LIN {X 0,Y 392.045,Z 91.25,A -85,B 0,C 180,E1 -11582.798,E2 -11582.798} C_VEL
LIN {X 0,Y 392.795,Z 97.506,A -85,B 0,C 180,E1 -11584.57,E2 -11584.57} C_VEL
LIN {X 0,Y 391.908,Z 107.771,A -85,B 0,C 180,E1 -11587.322,E2 -11587.322} C_VEL
LIN {X 0,Y 391.284,Z 115.559,A -85,B 0,C 180,E1 -11589.464,E2 -11589.464} C_VEL
LIN {X 0,Y 391.838,Z 118.711,A -85,B 0,C 180,E1 -11589.614,E2 -11589.614} C_VEL
LIN {X 0,Y 396.751,Z 145.759,A -85,B 0,C 180,E1 -11590.385,E2 -11590.385} C_VEL
LIN {X 0,Y 395.854,Z 220.432,A -85,B 0,C 180,E1 -11591.765,E2 -11591.765} C_VEL
LIN {X 0,Y 395.489,Z 230.328,A -85,B 0,C 180,E1 -11592.049,E2 -11592.049} C_VEL
LIN {X 0,Y 394.92,Z 240.302,A -85,B 0,C 180,E1 -11592.457,E2 -11592.457} C_VEL
LIN {X 0,Y 394.307,Z 250.666,A -85,B 0,C 180,E1 -11593.031,E2 -11593.031} C_VEL
LIN {X 0,Y 393.558,Z 259.797,A -85,B 0,C 180,E1 -11593.665,E2 -11593.665} C_VEL
LIN {X 0,Y 392.875,Z 268.795,A -85,B 0,C 180,E1 -11594.435,E2 -11594.435} C_VEL
LIN {X 0,Y 392.089,Z 277.523,A -85,B 0,C 180,E1 -11595.334,E2 -11595.334} C_VEL
LIN {X 0,Y 391.44,Z 285.346,A -85,B 0,C 180,E1 -11596.297,E2 -11596.297} C_VEL
LIN {X 0,Y 390.892,Z 292.141,A -85,B 0,C 180,E1 -11597.276,E2 -11597.276} C_VEL
LIN {X 0,Y 390.295,Z 298.342,A -85,B 0,C 180,E1 -11598.312,E2 -11598.312} C_VEL
LIN {X 0,Y 389.714,Z 304.879,A -85,B 0,C 180,E1 -11599.611,E2 -11599.611} C_VEL
LIN {X 0,Y 389.377,Z 309.381,A -85,B 0,C 180,E1 -11600.651,E2 -11600.651} C_VEL
LIN {X 0,Y 389.017,Z 314.872,A -85,B 0,C 180,E1 -11602.213,E2 -11602.213} C_VEL
LIN {X 0,Y 388.796,Z 319.196,A -85,B 0,C 180,E1 -11603.774,E2 -11603.774} C_VEL
LIN {X 0,Y 388.738,Z 321.563,A -85,B 0,C 180,E1 -11604.814,E2 -11604.814} C_VEL
LIN {X 0,Y 388.7,Z 323.362,A -85,B 0,C 180,E1 -11605.853,E2 -11605.853} C_VEL
LIN {X 0,Y 388.661,Z 325.805,A -85,B 0,C 180,E1 -11607.927,E2 -11607.927} C_VEL
LIN {X 0,Y 388.705,Z 326.395,A -85,B 0,C 180,E1 -11608.964,E2 -11608.964} C_VEL
LIN {X 0,Y 388.705,Z 326.395,A -85,B 0,C 180,E1 -11611.036,E2 -11611.036} C_VEL
LIN {X 0,Y 388.661,Z 325.805,A -85,B 0,C 180,E1 -11612.073,E2 -11612.073} C_VEL
LIN {X 0,Y 388.699,Z 323.362,A -85,B 0,C 180,E1 -11614.147,E2 -11614.147} C_VEL
LIN {X 0,Y 388.726,Z 320.312,A -85,B 0,C 180,E1 -11615.75,E2 -11615.75} C_VEL
LIN {X 0,Y 388.933,Z 316.426,A -85,B 0,C 180,E1 -11617.267,E2 -11617.267} C_VEL
LIN {X 0,Y 389.249,Z 311.297,A -85,B 0,C 180,E1 -11618.828,E2 -11618.828} C_VEL
LIN {X 0,Y 389.628,Z 306.034,A -85,B 0,C 180,E1 -11620.129,E2 -11620.129} C_VEL
LIN {X 0,Y 390.149,Z 299.717,A -85,B 0,C 180,E1 -11621.429,E2 -11621.429} C_VEL
LIN {X 0,Y 390.723,Z 293.767,A -85,B 0,C 180,E1 -11622.465,E2 -11622.465} C_VEL
LIN {X 0,Y 391.336,Z 286.839,A -85,B 0,C 180,E1 -11623.501,E2 -11623.501} C_VEL
LIN {X 0,Y 392.026,Z 278.658,A -85,B 0,C 180,E1 -11624.536,E2 -11624.536} C_VEL
LIN {X 0,Y 392.733,Z 270.146,A -85,B 0,C 180,E1 -11625.438,E2 -11625.438} C_VEL
LIN {X 0,Y 393.459,Z 261.43,A -85,B 0,C 180,E1 -11626.206,E2 -11626.206} C_VEL
LIN {X 0,Y 394.208,Z 251.672,A -85,B 0,C 180,E1 -11626.907,E2 -11626.907} C_VEL
LIN {X 0,Y 394.854,Z 241.59,A -85,B 0,C 180,E1 -11627.479,E2 -11627.479} C_VEL
LIN {X 0,Y 395.411,Z 232.076,A -85,B 0,C 180,E1 -11627.888,E2 -11627.888} C_VEL
LIN {X 0,Y 395.772,Z 221.762,A -85,B 0,C 180,E1 -11628.205,E2 -11628.205} C_VEL
LIN {X 0,Y 396.467,Z 173.837,A -85,B 0,C 180,E1 -11629.102,E2 -11629.102} C_VEL
LIN {X 0,Y 396.69,Z 145.088,A -85,B 0,C 180,E1 -11629.631,E2 -11629.631} C_VEL
LIN {X 0,Y 391.471,Z 116.921,A -85,B 0,C 180,E1 -11630.44,E2 -11630.44} C_VEL
LIN {X 0,Y 391.302,Z 115.351,A -85,B 0,C 180,E1 -11630.57,E2 -11630.57} C_VEL
LIN {X 0,Y 392.552,Z 100.812,A -85,B 0,C 180,E1 -11634.598,E2 -11634.598} C_VEL
LIN {X 0,Y 392.796,Z 95.971,A -85,B 0,C 180,E1 -11635.937,E2 -11635.937} C_VEL
LIN {X 0,Y 391.365,Z 87.664,A -85,B 0,C 180,E1 -11638.366,E2 -11638.366} C_VEL
LIN {X 0,Y 390.091,Z 81.417,A -85,B 0,C 180,E1 -11640.333,E2 -11640.333} C_VEL
LIN {X 0,Y 390.071,Z 81.395,A -85,B 0,C 180,E1 -11644.024,E2 -11644.024} C_VEL
LIN {X 0,Y 390.047,Z 81.402,A -85,B 0,C 180,E1 -11647.551,E2 -11647.551} C_VEL
LIN {X 0,Y 390.058,Z 81.38,A -85,B 0,C 180,E1 -11650.821,E2 -11650.821} C_VEL
LIN {X 0,Y 390.056,Z 81.396,A -85,B 0,C 180,E1 -11653.886,E2 -11653.886} C_VEL
LIN {X 0,Y 390.058,Z 81.396,A -85,B 0,C 180,E1 -11656.789,E2 -11656.789} C_VEL
LIN {X 0,Y 390.058,Z 81.388,A -85,B 0,C 180,E1 -11659.56,E2 -11659.56} C_VEL
LIN {X 0,Y 390.044,Z 81.398,A -85,B 0,C 180,E1 -11662.449,E2 -11662.449} C_VEL
LIN {X 0,Y 390.069,Z 81.38,A -85,B 0,C 180,E1 -11665.975,E2 -11665.975} C_VEL
LIN {X 0,Y 390.048,Z 81.396,A -85,B 0,C 180,E1 -11669.868,E2 -11669.868} C_VEL
LIN {X 0,Y 390.114,Z 81.372,A -85,B 0,C 180,E1 -11673.231,E2 -11673.231} C_VEL
LIN {X 0,Y 390.107,Z 81.393,A -85,B 0,C 180,E1 -11676.75,E2 -11676.75} C_VEL
LIN {X 0,Y 390.105,Z 81.378,A -85,B 0,C 180,E1 -11679.983,E2 -11679.983} C_VEL
LIN {X 0,Y 390.139,Z 81.378,A -85,B 0,C 180,E1 -11683.248,E2 -11683.248} C_VEL
LIN {X 0,Y 390.195,Z 81.377,A -85,B 0,C 180,E1 -11686.561,E2 -11686.561} C_VEL
LIN {X 0,Y 390.205,Z 81.355,A -85,B 0,C 180,E1 -11690.671,E2 -11690.671} C_VEL
LIN {X 0,Y 390.319,Z 81.359,A -85,B 0,C 180,E1 -11692.759,E2 -11692.759} C_VEL
LIN {X 0,Y 390.23,Z 81.374,A -85,B 0,C 180,E1 -11694.833,E2 -11694.833} C_VEL
LIN {X 0,Y 390.418,Z 81.341,A -85,B 0,C 180,E1 -11697.936,E2 -11697.936} C_VEL
LIN {X 0,Y 390.548,Z 81.311,A -85,B 0,C 180,E1 -11699.999,E2 -11699.999} C_VEL
LIN {X 0,Y 390.31,Z 81.358,A -85,B 0,C 180,E1 -11703.096,E2 -11703.096} C_VEL
LIN {X 0,Y 390.309,Z 81.36,A -85,B 0,C 180,E1 -11706.633,E2 -11706.633} C_VEL
LIN {X 0,Y 390.206,Z 81.356,A -85,B 0,C 180,E1 -11709.328,E2 -11709.328} C_VEL
LIN {X 0,Y 390.177,Z 81.375,A -85,B 0,C 180,E1 -11712.482,E2 -11712.482} C_VEL
LIN {X 0,Y 390.139,Z 81.385,A -85,B 0,C 180,E1 -11715.676,E2 -11715.676} C_VEL
LIN {X 0,Y 390.104,Z 81.37,A -85,B 0,C 180,E1 -11718.921,E2 -11718.921} C_VEL
LIN {X 0,Y 390.045,Z 81.395,A -85,B 0,C 180,E1 -11722.233,E2 -11722.233} C_VEL
LIN {X 0,Y 390.117,Z 81.379,A -85,B 0,C 180,E1 -11725.743,E2 -11725.743} C_VEL
LIN {X 0,Y 390.056,Z 81.391,A -85,B 0,C 180,E1 -11729.109,E2 -11729.109} C_VEL
LIN {X 0,Y 390.04,Z 81.396,A -85,B 0,C 180,E1 -11732.721,E2 -11732.721} C_VEL
LIN {X 0,Y 390.055,Z 81.391,A -85,B 0,C 180,E1 -11735.825,E2 -11735.825} C_VEL
LIN {X 0,Y 390.071,Z 81.39,A -85,B 0,C 180,E1 -11739.219,E2 -11739.219} C_VEL
LIN {X 0,Y 390.077,Z 81.392,A -85,B 0,C 180,E1 -11742.38,E2 -11742.38} C_VEL
LIN {X 0,Y 390.051,Z 81.378,A -85,B 0,C 180,E1 -11746.114,E2 -11746.114} C_VEL
LIN {X 0,Y 390.052,Z 81.381,A -85,B 0,C 180,E1 -11749.56,E2 -11749.56} C_VEL
LIN {X 0,Y 390.042,Z 81.4,A -85,B 0,C 180,E1 -11752.448,E2 -11752.448} C_VEL
LIN {X 0,Y 390.064,Z 81.374,A -85,B 0,C 180,E1 -11755.975,E2 -11755.975} C_VEL
LIN {X 0,Y 390.035,Z 81.39,A -85,B 0,C 180,E1 -11759.7,E2 -11759.7} C_VEL
LIN {X 0,Y 390.11,Z 81.392,A -85,B 0,C 180,E1 -11763.232,E2 -11763.232} C_VEL
LIN {X 0,Y 390.103,Z 81.393,A -85,B 0,C 180,E1 -11766.75,E2 -11766.75} C_VEL
LIN {X 0,Y 390.1,Z 81.395,A -85,B 0,C 180,E1 -11769.983,E2 -11769.983} C_VEL
LIN {X 0,Y 390.135,Z 81.391,A -85,B 0,C 180,E1 -11773.248,E2 -11773.248} C_VEL
LIN {X 0,Y 390.191,Z 81.383,A -85,B 0,C 180,E1 -11776.561,E2 -11776.561} C_VEL
LIN {X 0,Y 390.202,Z 81.382,A -85,B 0,C 180,E1 -11780.671,E2 -11780.671} C_VEL
LIN {X 0,Y 390.404,Z 81.767,A -85,B 0,C 180,E1 -11781.927,E2 -11781.927} C_VEL
LIN {X 0,Y 391.193,Z 83.981,A -85,B 0,C 180,E1 -11782.905,E2 -11782.905} C_VEL
LIN {X 0,Y 392.561,Z 85.719,A -85,B 0,C 180,E1 -11783.962,E2 -11783.962} C_VEL
LIN {X 0,Y 394.309,Z 87.002,A -85,B 0,C 180,E1 -11785.656,E2 -11785.656} C_VEL
LIN {X 0,Y 395.582,Z 87.492,A -85,B 0,C 180,E1 -11787.454,E2 -11787.454} C_VEL
LIN {X 0,Y 396.184,Z 87.941,A -85,B 0,C 180,E1 -11788.984,E2 -11788.984} C_VEL
LIN {X 0,Y 396.323,Z 87.848,A -85,B 0,C 180,E1 -11790,E2 -11790} C_VEL
LIN {X 0,Y 396.07,Z 87.804,A -85,B 0,C 180,E1 -11791.525,E2 -11791.525} C_VEL
LIN {X 0,Y 395.354,Z 87.371,A -85,B 0,C 180,E1 -11793.057,E2 -11793.057} C_VEL
LIN {X 0,Y 393.693,Z 86.657,A -85,B 0,C 180,E1 -11794.993,E2 -11794.993} C_VEL
LIN {X 0,Y 391.897,Z 85.017,A -85,B 0,C 180,E1 -11796.565,E2 -11796.565} C_VEL
LIN {X 0,Y 390.579,Z 82.501,A -85,B 0,C 180,E1 -11797.684,E2 -11797.684} C_VEL
LIN {X 0,Y 390.341,Z 81.593,A -85,B 0,C 180,E1 -11798.282,E2 -11798.282} C_VEL
LIN {X 0,Y 390.145,Z 81.389,A -85,B 0,C 180,E1 -11801.429,E2 -11801.429} C_VEL
LIN {X 0,Y 390.141,Z 81.39,A -85,B 0,C 180,E1 -11804.607,E2 -11804.607} C_VEL
LIN {X 0,Y 390.125,Z 81.392,A -85,B 0,C 180,E1 -11807.833,E2 -11807.833} C_VEL
LIN {X 0,Y 390.052,Z 81.4,A -85,B 0,C 180,E1 -11811.122,E2 -11811.122} C_VEL
LIN {X 0,Y 390.077,Z 81.398,A -85,B 0,C 180,E1 -11814.481,E2 -11814.481} C_VEL
LIN {X 0,Y 390.113,Z 81.386,A -85,B 0,C 180,E1 -11817.93,E2 -11817.93} C_VEL
LIN {X 0,Y 390.009,Z 81.395,A -85,B 0,C 180,E1 -11820.802,E2 -11820.802} C_VEL
LIN {X 0,Y 389.336,Z 81.489,A -85,B 0,C 180,E1 -11821.664,E2 -11821.664} C_VEL
LIN {X 0,Y 386.489,Z 81.835,A -85,B 0,C 180,E1 -11823.066,E2 -11823.066} C_VEL
LIN {X 0,Y 384.09,Z 82.119,A -85,B 0,C 180,E1 -11824.199,E2 -11824.199} C_VEL
LIN {X 0,Y 383.072,Z 82.24,A -85,B 0,C 180,E1 -11825.075,E2 -11825.075} C_VEL
LIN {X 0,Y 382.995,Z 82.252,A -85,B 0,C 180,E1 -11825.371,E2 -11825.371} C_VEL
LIN {X 0,Y 383.002,Z 82.275,A -85,B 0,C 180,E1 -11828.601,E2 -11828.601} C_VEL
LIN {X 0,Y 382.979,Z 82.245,A -85,B 0,C 180,E1 -11831.348,E2 -11831.348} C_VEL
LIN {X 0,Y 382.992,Z 82.265,A -85,B 0,C 180,E1 -11834.304,E2 -11834.304} C_VEL
LIN {X 0,Y 383.036,Z 82.275,A -85,B 0,C 180,E1 -11837.245,E2 -11837.245} C_VEL
LIN {X 0,Y 383.018,Z 82.267,A -85,B 0,C 180,E1 -11840.413,E2 -11840.413} C_VEL
LIN {X 0,Y 383.024,Z 82.267,A -85,B 0,C 180,E1 -11844.045,E2 -11844.045} C_VEL
LIN {X 0,Y 382.984,Z 82.278,A -85,B 0,C 180,E1 -11847.578,E2 -11847.578} C_VEL
LIN {X 0,Y 382.99,Z 82.275,A -85,B 0,C 180,E1 -11850.301,E2 -11850.301} C_VEL
LIN {X 0,Y 383.078,Z 82.254,A -85,B 0,C 180,E1 -11854.021,E2 -11854.021} C_VEL
LIN {X 0,Y 383.011,Z 82.273,A -85,B 0,C 180,E1 -11857.336,E2 -11857.336} C_VEL
LIN {X 0,Y 383.059,Z 82.247,A -85,B 0,C 180,E1 -11860.717,E2 -11860.717} C_VEL
LIN {X 0,Y 383.08,Z 82.261,A -85,B 0,C 180,E1 -11864.027,E2 -11864.027} C_VEL
LIN {X 0,Y 383.14,Z 82.252,A -85,B 0,C 180,E1 -11867.285,E2 -11867.285} C_VEL
LIN {X 0,Y 383.152,Z 82.233,A -85,B 0,C 180,E1 -11870.499,E2 -11870.499} C_VEL
LIN {X 0,Y 383.273,Z 82.236,A -85,B 0,C 180,E1 -11872.626,E2 -11872.626} C_VEL
LIN {X 0,Y 383.198,Z 82.251,A -85,B 0,C 180,E1 -11874.739,E2 -11874.739} C_VEL
LIN {X 0,Y 383.385,Z 82.216,A -85,B 0,C 180,E1 -11877.899,E2 -11877.899} C_VEL
LIN {X 0,Y 383.517,Z 82.186,A -85,B 0,C 180,E1 -11880.001,E2 -11880.001} C_VEL
LIN {X 0,Y 383.246,Z 82.24,A -85,B 0,C 180,E1 -11883.154,E2 -11883.154} C_VEL
LIN {X 0,Y 383.294,Z 82.235,A -85,B 0,C 180,E1 -11886.317,E2 -11886.317} C_VEL
LIN {X 0,Y 383.26,Z 82.223,A -85,B 0,C 180,E1 -11888.436,E2 -11888.436} C_VEL
LIN {X 0,Y 383.097,Z 82.25,A -85,B 0,C 180,E1 -11891.643,E2 -11891.643} C_VEL
LIN {X 0,Y 383.111,Z 82.259,A -85,B 0,C 180,E1 -11894.882,E2 -11894.882} C_VEL
LIN {X 0,Y 383.063,Z 82.243,A -85,B 0,C 180,E1 -11898.174,E2 -11898.174} C_VEL
LIN {X 0,Y 383,Z 82.272,A -85,B 0,C 180,E1 -11901.531,E2 -11901.531} C_VEL
LIN {X 0,Y 383.053,Z 82.264,A -85,B 0,C 180,E1 -11904.961,E2 -11904.961} C_VEL
LIN {X 0,Y 383.031,Z 82.26,A -85,B 0,C 180,E1 -11908.271,E2 -11908.271} C_VEL
LIN {X 0,Y 383.01,Z 82.272,A -85,B 0,C 180,E1 -11912.15,E2 -11912.15} C_VEL
LIN {X 0,Y 383.019,Z 82.259,A -85,B 0,C 180,E1 -11914.668,E2 -11914.668} C_VEL
LIN {X 0,Y 383,Z 82.275,A -85,B 0,C 180,E1 -11917.904,E2 -11917.904} C_VEL
LIN {X 0,Y 382.985,Z 82.276,A -85,B 0,C 180,E1 -11921.348,E2 -11921.348} C_VEL
LIN {X 0,Y 382.997,Z 82.273,A -85,B 0,C 180,E1 -11924.304,E2 -11924.304} C_VEL
LIN {X 0,Y 383.012,Z 82.273,A -85,B 0,C 180,E1 -11927.241,E2 -11927.241} C_VEL
LIN {X 0,Y 383.017,Z 82.255,A -85,B 0,C 180,E1 -11930.414,E2 -11930.414} C_VEL
LIN {X 0,Y 383.029,Z 82.263,A -85,B 0,C 180,E1 -11934.045,E2 -11934.045} C_VEL
LIN {X 0,Y 382.989,Z 82.271,A -85,B 0,C 180,E1 -11937.578,E2 -11937.578} C_VEL
LIN {X 0,Y 383.078,Z 82.492,A -85,B 0,C 180,E1 -11939.465,E2 -11939.465} C_VEL
LIN {X 0,Y 385.01,Z 92.117,A -85,B 0,C 180,E1 -11942.554,E2 -11942.554} C_VEL
LIN {X 0,Y 385.816,Z 98.375,A -85,B 0,C 180,E1 -11944.366,E2 -11944.366} C_VEL
LIN {X 0,Y 385.017,Z 107.585,A -85,B 0,C 180,E1 -11946.893,E2 -11946.893} C_VEL
LIN {X 0,Y 384.386,Z 115.368,A -85,B 0,C 180,E1 -11949.077,E2 -11949.077} C_VEL
LIN {X 0,Y 384.801,Z 117.965,A -85,B 0,C 180,E1 -11949.214,E2 -11949.214} C_VEL
LIN {X 0,Y 389.753,Z 144.646,A -85,B 0,C 180,E1 -11950,E2 -11950} C_VEL
LIN {X 0,Y 390.081,Z 149.092,A -85,B 0,C 180,E1 -11950.103,E2 -11950.103} C_VEL
LIN {X 0,Y 389.104,Z 220.241,A -85,B 0,C 180,E1 -11951.437,E2 -11951.437} C_VEL
LIN {X 0,Y 388.732,Z 230.137,A -85,B 0,C 180,E1 -11951.726,E2 -11951.726} C_VEL
LIN {X 0,Y 388.163,Z 240.112,A -85,B 0,C 180,E1 -11952.142,E2 -11952.142} C_VEL
LIN {X 0,Y 387.602,Z 249.468,A -85,B 0,C 180,E1 -11952.66,E2 -11952.66} C_VEL
LIN {X 0,Y 386.761,Z 259.607,A -85,B 0,C 180,E1 -11953.369,E2 -11953.369} C_VEL
LIN {X 0,Y 386.012,Z 268.604,A -85,B 0,C 180,E1 -11954.151,E2 -11954.151} C_VEL
LIN {X 0,Y 385.218,Z 277.332,A -85,B 0,C 180,E1 -11955.066,E2 -11955.066} C_VEL
LIN {X 0,Y 384.497,Z 285.33,A -85,B 0,C 180,E1 -11956.069,E2 -11956.069} C_VEL
LIN {X 0,Y 383.783,Z 293.576,A -85,B 0,C 180,E1 -11957.306,E2 -11957.306} C_VEL
LIN {X 0,Y 383.168,Z 299.526,A -85,B 0,C 180,E1 -11958.36,E2 -11958.36} C_VEL
LIN {X 0,Y 382.609,Z 305.843,A -85,B 0,C 180,E1 -11959.683,E2 -11959.683} C_VEL
LIN {X 0,Y 382.204,Z 311.106,A -85,B 0,C 180,E1 -11961.008,E2 -11961.008} C_VEL
LIN {X 0,Y 381.861,Z 316.235,A -85,B 0,C 180,E1 -11962.598,E2 -11962.598} C_VEL
LIN {X 0,Y 381.688,Z 319.523,A -85,B 0,C 180,E1 -11963.883,E2 -11963.883} C_VEL
LIN {X 0,Y 381.639,Z 321.372,A -85,B 0,C 180,E1 -11964.717,E2 -11964.717} C_VEL
LIN {X 0,Y 381.625,Z 323.171,A -85,B 0,C 180,E1 -11965.776,E2 -11965.776} C_VEL
LIN {X 0,Y 381.56,Z 325.614,A -85,B 0,C 180,E1 -11967.889,E2 -11967.889} C_VEL
LIN {X 0,Y 381.604,Z 326.204,A -85,B 0,C 180,E1 -11968.945,E2 -11968.945} C_VEL
LIN {X 0,Y 381.604,Z 326.204,A -85,B 0,C 180,E1 -11971.055,E2 -11971.055} C_VEL
LIN {X 0,Y 381.56,Z 325.614,A -85,B 0,C 180,E1 -11972.111,E2 -11972.111} C_VEL
LIN {X 0,Y 381.625,Z 323.171,A -85,B 0,C 180,E1 -11974.224,E2 -11974.224} C_VEL
LIN {X 0,Y 381.639,Z 321.372,A -85,B 0,C 180,E1 -11975.283,E2 -11975.283} C_VEL
LIN {X 0,Y 381.781,Z 317.765,A -85,B 0,C 180,E1 -11976.872,E2 -11976.872} C_VEL
LIN {X 0,Y 382.057,Z 313.021,A -85,B 0,C 180,E1 -11978.462,E2 -11978.462} C_VEL
LIN {X 0,Y 382.507,Z 306.999,A -85,B 0,C 180,E1 -11980.052,E2 -11980.052} C_VEL
LIN {X 0,Y 383.045,Z 300.902,A -85,B 0,C 180,E1 -11981.375,E2 -11981.375} C_VEL
LIN {X 0,Y 383.624,Z 295.203,A -85,B 0,C 180,E1 -11982.431,E2 -11982.431} C_VEL
LIN {X 0,Y 384.396,Z 286.648,A -85,B 0,C 180,E1 -11983.75,E2 -11983.75} C_VEL
LIN {X 0,Y 385.147,Z 278.468,A -85,B 0,C 180,E1 -11984.801,E2 -11984.801} C_VEL
LIN {X 0,Y 385.886,Z 269.955,A -85,B 0,C 180,E1 -11985.719,E2 -11985.719} C_VEL
LIN {X 0,Y 386.631,Z 261.239,A -85,B 0,C 180,E1 -11986.5,E2 -11986.5} C_VEL
LIN {X 0,Y 387.407,Z 251.481,A -85,B 0,C 180,E1 -11987.213,E2 -11987.213} C_VEL
LIN {X 0,Y 388.099,Z 241.4,A -85,B 0,C 180,E1 -11987.793,E2 -11987.793} C_VEL
LIN {X 0,Y 388.629,Z 231.885,A -85,B 0,C 180,E1 -11988.211,E2 -11988.211} C_VEL
LIN {X 0,Y 389.027,Z 221.572,A -85,B 0,C 180,E1 -11988.532,E2 -11988.532} C_VEL
LIN {X 0,Y 389.708,Z 180.023,A -85,B 0,C 180,E1 -11989.325,E2 -11989.325} C_VEL
LIN {X 0,Y 389.993,Z 145.947,A -85,B 0,C 180,E1 -11989.962,E2 -11989.962} C_VEL
LIN {X 0,Y 384.773,Z 117.818,A -85,B 0,C 180,E1 -11990.791,E2 -11990.791} C_VEL
LIN {X 0,Y 384.356,Z 115.382,A -85,B 0,C 180,E1 -11990.921,E2 -11990.921} C_VEL
LIN {X 0,Y 385.625,Z 101.633,A -85,B 0,C 180,E1 -11994.782,E2 -11994.782} C_VEL
LIN {X 0,Y 385.861,Z 97.629,A -85,B 0,C 180,E1 -11995.921,E2 -11995.921} C_VEL
LIN {X 0,Y 384.672,Z 90.41,A -85,B 0,C 180,E1 -11998.064,E2 -11998.064} C_VEL
LIN {X 0,Y 383.05,Z 82.333,A -85,B 0,C 180,E1 -12000.617,E2 -12000.617} C_VEL
LIN {X 0,Y 383.02,Z 82.27,A -85,B 0,C 180,E1 -12004.34,E2 -12004.34} C_VEL
LIN {X 0,Y 382.999,Z 82.277,A -85,B 0,C 180,E1 -12007.268,E2 -12007.268} C_VEL
LIN {X 0,Y 383.01,Z 82.254,A -85,B 0,C 180,E1 -12009.958,E2 -12009.958} C_VEL
LIN {X 0,Y 383.007,Z 82.274,A -85,B 0,C 180,E1 -12012.778,E2 -12012.778} C_VEL
LIN {X 0,Y 382.999,Z 82.274,A -85,B 0,C 180,E1 -12015.789,E2 -12015.789} C_VEL
LIN {X 0,Y 382.99,Z 82.276,A -85,B 0,C 180,E1 -12018.795,E2 -12018.795} C_VEL
LIN {X 0,Y 383,Z 82.275,A -85,B 0,C 180,E1 -12022.096,E2 -12022.096} C_VEL
LIN {X 0,Y 383.019,Z 82.259,A -85,B 0,C 180,E1 -12025.332,E2 -12025.332} C_VEL
LIN {X 0,Y 382.984,Z 82.281,A -85,B 0,C 180,E1 -12029.081,E2 -12029.081} C_VEL
LIN {X 0,Y 383.058,Z 82.251,A -85,B 0,C 180,E1 -12032.698,E2 -12032.698} C_VEL
LIN {X 0,Y 383.053,Z 82.264,A -85,B 0,C 180,E1 -12035.039,E2 -12035.039} C_VEL
LIN {X 0,Y 383,Z 82.272,A -85,B 0,C 180,E1 -12038.469,E2 -12038.469} C_VEL
LIN {X 0,Y 383.063,Z 82.243,A -85,B 0,C 180,E1 -12041.826,E2 -12041.826} C_VEL
LIN {X 0,Y 383.111,Z 82.259,A -85,B 0,C 180,E1 -12045.118,E2 -12045.118} C_VEL
LIN {X 0,Y 383.097,Z 82.25,A -85,B 0,C 180,E1 -12048.357,E2 -12048.357} C_VEL
LIN {X 0,Y 383.304,Z 82.221,A -85,B 0,C 180,E1 -12051.932,E2 -12051.932} C_VEL
LIN {X 0,Y 383.202,Z 82.25,A -85,B 0,C 180,E1 -12054.738,E2 -12054.738} C_VEL
LIN {X 0,Y 383.385,Z 82.217,A -85,B 0,C 180,E1 -12057.898,E2 -12057.898} C_VEL
LIN {X 0,Y 383.517,Z 82.186,A -85,B 0,C 180,E1 -12059.999,E2 -12059.999} C_VEL
LIN {X 0,Y 383.246,Z 82.238,A -85,B 0,C 180,E1 -12063.153,E2 -12063.153} C_VEL
LIN {X 0,Y 383.269,Z 82.236,A -85,B 0,C 180,E1 -12066.627,E2 -12066.627} C_VEL
LIN {X 0,Y 383.259,Z 82.226,A -85,B 0,C 180,E1 -12068.435,E2 -12068.435} C_VEL
LIN {X 0,Y 383.106,Z 82.249,A -85,B 0,C 180,E1 -12071.641,E2 -12071.641} C_VEL
LIN {X 0,Y 383.111,Z 82.262,A -85,B 0,C 180,E1 -12074.881,E2 -12074.881} C_VEL
LIN {X 0,Y 383.061,Z 82.248,A -85,B 0,C 180,E1 -12078.173,E2 -12078.173} C_VEL
LIN {X 0,Y 382.997,Z 82.273,A -85,B 0,C 180,E1 -12081.53,E2 -12081.53} C_VEL
LIN {X 0,Y 383.05,Z 82.267,A -85,B 0,C 180,E1 -12084.96,E2 -12084.96} C_VEL
LIN {X 0,Y 383.027,Z 82.258,A -85,B 0,C 180,E1 -12088.27,E2 -12088.27} C_VEL
LIN {X 0,Y 383.007,Z 82.274,A -85,B 0,C 180,E1 -12092.149,E2 -12092.149} C_VEL
LIN {X 0,Y 383.015,Z 82.261,A -85,B 0,C 180,E1 -12094.667,E2 -12094.667} C_VEL
LIN {X 0,Y 383,Z 82.276,A -85,B 0,C 180,E1 -12097.904,E2 -12097.904} C_VEL
LIN {X 0,Y 383.01,Z 82.269,A -85,B 0,C 180,E1 -12101.343,E2 -12101.343} C_VEL
LIN {X 0,Y 382.993,Z 82.277,A -85,B 0,C 180,E1 -12104.303,E2 -12104.303} C_VEL
LIN {X 0,Y 383.006,Z 82.241,A -85,B 0,C 180,E1 -12107.24,E2 -12107.24} C_VEL
LIN {X 0,Y 383.012,Z 82.265,A -85,B 0,C 180,E1 -12110.413,E2 -12110.413} C_VEL
LIN {X 0,Y 383.023,Z 82.258,A -85,B 0,C 180,E1 -12114.044,E2 -12114.044} C_VEL
LIN {X 0,Y 382.983,Z 82.276,A -85,B 0,C 180,E1 -12117.578,E2 -12117.578} C_VEL
LIN {X 0,Y 382.988,Z 82.262,A -85,B 0,C 180,E1 -12120.3,E2 -12120.3} C_VEL
LIN {X 0,Y 383.077,Z 82.27,A -85,B 0,C 180,E1 -12124.021,E2 -12124.021} C_VEL
LIN {X 0,Y 383.005,Z 82.278,A -85,B 0,C 180,E1 -12127.335,E2 -12127.335} C_VEL
LIN {X 0,Y 383.057,Z 82.271,A -85,B 0,C 180,E1 -12130.716,E2 -12130.716} C_VEL
LIN {X 0,Y 383.077,Z 82.269,A -85,B 0,C 180,E1 -12134.027,E2 -12134.027} C_VEL
LIN {X 0,Y 383.133,Z 82.262,A -85,B 0,C 180,E1 -12137.284,E2 -12137.284} C_VEL
LIN {X 0,Y 383.161,Z 82.567,A -85,B 0,C 180,E1 -12138.561,E2 -12138.561} C_VEL
LIN {X 0,Y 383.436,Z 83.716,A -85,B 0,C 180,E1 -12138.971,E2 -12138.971} C_VEL
LIN {X 0,Y 384.578,Z 85.76,A -85,B 0,C 180,E1 -12139.603,E2 -12139.603} C_VEL
LIN {X 0,Y 386.856,Z 87.64,A -85,B 0,C 180,E1 -12140.722,E2 -12140.722} C_VEL
LIN {X 0,Y 388.921,Z 88.829,A -85,B 0,C 180,E1 -12141.896,E2 -12141.896} C_VEL
LIN {X 0,Y 390.34,Z 91.395,A -85,B 0,C 180,E1 -12142.955,E2 -12142.955} C_VEL
LIN {X 0,Y 391.933,Z 93.07,A -85,B 0,C 180,E1 -12144.211,E2 -12144.211} C_VEL
LIN {X 0,Y 393.437,Z 94.033,A -85,B 0,C 180,E1 -12145.646,E2 -12145.646} C_VEL
LIN {X 0,Y 394.719,Z 94.512,A -85,B 0,C 180,E1 -12147.449,E2 -12147.449} C_VEL
LIN {X 0,Y 395.318,Z 94.987,A -85,B 0,C 180,E1 -12148.981,E2 -12148.981} C_VEL
LIN {X 0,Y 395.458,Z 94.896,A -85,B 0,C 180,E1 -12150,E2 -12150} C_VEL
LIN {X 0,Y 395.202,Z 94.853,A -85,B 0,C 180,E1 -12151.529,E2 -12151.529} C_VEL
LIN {X 0,Y 394.244,Z 94.355,A -85,B 0,C 180,E1 -12153.368,E2 -12153.368} C_VEL
LIN {X 0,Y 392.65,Z 93.62,A -85,B 0,C 180,E1 -12155.135,E2 -12155.135} C_VEL
LIN {X 0,Y 390.975,Z 92.169,A -85,B 0,C 180,E1 -12156.58,E2 -12156.58} C_VEL
LIN {X 0,Y 389.337,Z 89.59,A -85,B 0,C 180,E1 -12157.841,E2 -12157.841} C_VEL
LIN {X 0,Y 388.549,Z 88.461,A -85,B 0,C 180,E1 -12158.32,E2 -12158.32} C_VEL
LIN {X 0,Y 385.836,Z 87.007,A -85,B 0,C 180,E1 -12159.766,E2 -12159.766} C_VEL
LIN {X 0,Y 383.934,Z 84.789,A -85,B 0,C 180,E1 -12160.748,E2 -12160.748} C_VEL
LIN {X 0,Y 383.222,Z 82.963,A -85,B 0,C 180,E1 -12161.236,E2 -12161.236} C_VEL
LIN {X 0,Y 383.115,Z 82.297,A -85,B 0,C 180,E1 -12161.91,E2 -12161.91} C_VEL
LIN {X 0,Y 383.107,Z 82.266,A -85,B 0,C 180,E1 -12164.882,E2 -12164.882} C_VEL
LIN {X 0,Y 383.086,Z 82.268,A -85,B 0,C 180,E1 -12168.172,E2 -12168.172} C_VEL
LIN {X 0,Y 382.99,Z 82.28,A -85,B 0,C 180,E1 -12171.531,E2 -12171.531} C_VEL
LIN {X 0,Y 383.049,Z 82.271,A -85,B 0,C 180,E1 -12174.96,E2 -12174.96} C_VEL
LIN {X 0,Y 383.013,Z 82.262,A -85,B 0,C 180,E1 -12178.495,E2 -12178.495} C_VEL
LIN {X 0,Y 383.008,Z 82.276,A -85,B 0,C 180,E1 -12182.15,E2 -12182.15} C_VEL
LIN {X 0,Y 382.995,Z 82.252,A -85,B 0,C 180,E1 -12185.371,E2 -12185.371} C_VEL
LIN {X 0,Y 382.359,Z 82.347,A -85,B 0,C 180,E1 -12186.249,E2 -12186.249} C_VEL
LIN {X 0,Y 379.564,Z 82.707,A -85,B 0,C 180,E1 -12187.677,E2 -12187.677} C_VEL
LIN {X 0,Y 377.159,Z 83.005,A -85,B 0,C 180,E1 -12188.832,E2 -12188.832} C_VEL
LIN {X 0,Y 376.087,Z 83.127,A -85,B 0,C 180,E1 -12189.724,E2 -12189.724} C_VEL
LIN {X 0,Y 375.98,Z 83.135,A -85,B 0,C 180,E1 -12190.026,E2 -12190.026} C_VEL
LIN {X 0,Y 375.925,Z 83.133,A -85,B 0,C 180,E1 -12193.766,E2 -12193.766} C_VEL
LIN {X 0,Y 375.957,Z 83.15,A -85,B 0,C 180,E1 -12197.704,E2 -12197.704} C_VEL
LIN {X 0,Y 375.965,Z 83.146,A -85,B 0,C 180,E1 -12200.539,E2 -12200.539} C_VEL
LIN {X 0,Y 375.962,Z 83.15,A -85,B 0,C 180,E1 -12203.496,E2 -12203.496} C_VEL
LIN {X 0,Y 375.957,Z 83.14,A -85,B 0,C 180,E1 -12205.889,E2 -12205.889} C_VEL
LIN {X 0,Y 375.962,Z 83.151,A -85,B 0,C 180,E1 -12209.688,E2 -12209.688} C_VEL
LIN {X 0,Y 376.017,Z 83.13,A -85,B 0,C 180,E1 -12213.348,E2 -12213.348} C_VEL
LIN {X 0,Y 375.996,Z 83.151,A -85,B 0,C 180,E1 -12216.889,E2 -12216.889} C_VEL
LIN {X 0,Y 375.996,Z 83.128,A -85,B 0,C 180,E1 -12220.34,E2 -12220.34} C_VEL
LIN {X 0,Y 376.028,Z 83.138,A -85,B 0,C 180,E1 -12223.719,E2 -12223.719} C_VEL
LIN {X 0,Y 376.106,Z 83.129,A -85,B 0,C 180,E1 -12227.043,E2 -12227.043} C_VEL
LIN {X 0,Y 376.12,Z 83.107,A -85,B 0,C 180,E1 -12230.319,E2 -12230.319} C_VEL
LIN {X 0,Y 376.23,Z 83.11,A -85,B 0,C 180,E1 -12232.487,E2 -12232.487} C_VEL
LIN {X 0,Y 376.171,Z 83.127,A -85,B 0,C 180,E1 -12234.64,E2 -12234.64} C_VEL
LIN {X 0,Y 376.351,Z 83.092,A -85,B 0,C 180,E1 -12237.86,E2 -12237.86} C_VEL
LIN {X 0,Y 376.487,Z 83.06,A -85,B 0,C 180,E1 -12240.001,E2 -12240.001} C_VEL
LIN {X 0,Y 376.185,Z 83.119,A -85,B 0,C 180,E1 -12243.214,E2 -12243.214} C_VEL
LIN {X 0,Y 376.252,Z 83.111,A -85,B 0,C 180,E1 -12246.435,E2 -12246.435} C_VEL
LIN {X 0,Y 376.206,Z 83.101,A -85,B 0,C 180,E1 -12248.596,E2 -12248.596} C_VEL
LIN {X 0,Y 376.05,Z 83.13,A -85,B 0,C 180,E1 -12251.864,E2 -12251.864} C_VEL
LIN {X 0,Y 376.059,Z 83.14,A -85,B 0,C 180,E1 -12255.168,E2 -12255.168} C_VEL
LIN {X 0,Y 376.009,Z 83.121,A -85,B 0,C 180,E1 -12258.527,E2 -12258.527} C_VEL
LIN {X 0,Y 375.969,Z 83.149,A -85,B 0,C 180,E1 -12261.954,E2 -12261.954} C_VEL
LIN {X 0,Y 376.007,Z 83.134,A -85,B 0,C 180,E1 -12265.462,E2 -12265.462} C_VEL
LIN {X 0,Y 375.962,Z 83.147,A -85,B 0,C 180,E1 -12269.08,E2 -12269.08} C_VEL
LIN {X 0,Y 375.95,Z 83.146,A -85,B 0,C 180,E1 -12272.829,E2 -12272.829} C_VEL
LIN {X 0,Y 375.959,Z 83.147,A -85,B 0,C 180,E1 -12275.416,E2 -12275.416} C_VEL
LIN {X 0,Y 375.974,Z 83.152,A -85,B 0,C 180,E1 -12278.271,E2 -12278.271} C_VEL
LIN {X 0,Y 375.936,Z 83.154,A -85,B 0,C 180,E1 -12281.601,E2 -12281.601} C_VEL
LIN {X 0,Y 375.928,Z 83.153,A -85,B 0,C 180,E1 -12285.269,E2 -12285.269} C_VEL
LIN {X 0,Y 375.936,Z 83.145,A -85,B 0,C 180,E1 -12288.4,E2 -12288.4} C_VEL
LIN {X 0,Y 375.977,Z 83.148,A -85,B 0,C 180,E1 -12291.73,E2 -12291.73} C_VEL
LIN {X 0,Y 375.982,Z 83.141,A -85,B 0,C 180,E1 -12295.333,E2 -12295.333} C_VEL
LIN {X 0,Y 375.989,Z 83.252,A -85,B 0,C 180,E1 -12299.095,E2 -12299.095} C_VEL
LIN {X 0,Y 377.574,Z 91.051,A -85,B 0,C 180,E1 -12301.71,E2 -12301.71} C_VEL
LIN {X 0,Y 378.775,Z 98.203,A -85,B 0,C 180,E1 -12303.853,E2 -12303.853} C_VEL
LIN {X 0,Y 378.644,Z 102.91,A -85,B 0,C 180,E1 -12305.179,E2 -12305.179} C_VEL
LIN {X 0,Y 377.47,Z 115.277,A -85,B 0,C 180,E1 -12308.692,E2 -12308.692} C_VEL
LIN {X 0,Y 378.441,Z 120.426,A -85,B 0,C 180,E1 -12308.901,E2 -12308.901} C_VEL
LIN {X 0,Y 383.173,Z 146.01,A -85,B 0,C 180,E1 -12309.672,E2 -12309.672} C_VEL
LIN {X 0,Y 383.381,Z 153.964,A -85,B 0,C 180,E1 -12309.839,E2 -12309.839} C_VEL
LIN {X 0,Y 382.394,Z 220.051,A -85,B 0,C 180,E1 -12311.099,E2 -12311.099} C_VEL
LIN {X 0,Y 381.965,Z 230.821,A -85,B 0,C 180,E1 -12311.425,E2 -12311.425} C_VEL
LIN {X 0,Y 381.411,Z 239.921,A -85,B 0,C 180,E1 -12311.814,E2 -12311.814} C_VEL
LIN {X 0,Y 380.834,Z 249.278,A -85,B 0,C 180,E1 -12312.342,E2 -12312.342} C_VEL
LIN {X 0,Y 379.964,Z 259.416,A -85,B 0,C 180,E1 -12313.063,E2 -12313.063} C_VEL
LIN {X 0,Y 379.188,Z 268.413,A -85,B 0,C 180,E1 -12313.858,E2 -12313.858} C_VEL
LIN {X 0,Y 378.348,Z 277.141,A -85,B 0,C 180,E1 -12314.789,E2 -12314.789} C_VEL
LIN {X 0,Y 377.571,Z 285.301,A -85,B 0,C 180,E1 -12315.831,E2 -12315.831} C_VEL
LIN {X 0,Y 376.829,Z 293.385,A -85,B 0,C 180,E1 -12317.067,E2 -12317.067} C_VEL
LIN {X 0,Y 376.199,Z 299.335,A -85,B 0,C 180,E1 -12318.141,E2 -12318.141} C_VEL
LIN {X 0,Y 375.595,Z 305.652,A -85,B 0,C 180,E1 -12319.488,E2 -12319.488} C_VEL
LIN {X 0,Y 375.16,Z 310.914,A -85,B 0,C 180,E1 -12320.838,E2 -12320.838} C_VEL
LIN {X 0,Y 374.794,Z 316.044,A -85,B 0,C 180,E1 -12322.458,E2 -12322.458} C_VEL
LIN {X 0,Y 374.583,Z 319.714,A -85,B 0,C 180,E1 -12323.936,E2 -12323.936} C_VEL
LIN {X 0,Y 374.529,Z 322.98,A -85,B 0,C 180,E1 -12325.695,E2 -12325.695} C_VEL
LIN {X 0,Y 374.459,Z 325.424,A -85,B 0,C 180,E1 -12327.849,E2 -12327.849} C_VEL
LIN {X 0,Y 374.504,Z 326.013,A -85,B 0,C 180,E1 -12328.925,E2 -12328.925} C_VEL
LIN {X 0,Y 374.504,Z 326.013,A -85,B 0,C 180,E1 -12331.075,E2 -12331.075} C_VEL
LIN {X 0,Y 374.459,Z 325.424,A -85,B 0,C 180,E1 -12332.151,E2 -12332.151} C_VEL
LIN {X 0,Y 374.529,Z 322.98,A -85,B 0,C 180,E1 -12334.305,E2 -12334.305} C_VEL
LIN {X 0,Y 374.582,Z 319.714,A -85,B 0,C 180,E1 -12336.063,E2 -12336.063} C_VEL
LIN {X 0,Y 374.794,Z 316.044,A -85,B 0,C 180,E1 -12337.542,E2 -12337.542} C_VEL
LIN {X 0,Y 375.16,Z 310.914,A -85,B 0,C 180,E1 -12339.162,E2 -12339.162} C_VEL
LIN {X 0,Y 375.595,Z 305.652,A -85,B 0,C 180,E1 -12340.512,E2 -12340.512} C_VEL
LIN {X 0,Y 376.198,Z 299.335,A -85,B 0,C 180,E1 -12341.859,E2 -12341.859} C_VEL
LIN {X 0,Y 376.827,Z 293.385,A -85,B 0,C 180,E1 -12342.933,E2 -12342.933} C_VEL
LIN {X 0,Y 377.609,Z 285.248,A -85,B 0,C 180,E1 -12344.175,E2 -12344.175} C_VEL
LIN {X 0,Y 378.373,Z 277.142,A -85,B 0,C 180,E1 -12345.21,E2 -12345.21} C_VEL
LIN {X 0,Y 379.159,Z 268.412,A -85,B 0,C 180,E1 -12346.143,E2 -12346.143} C_VEL
LIN {X 0,Y 379.995,Z 259.417,A -85,B 0,C 180,E1 -12346.935,E2 -12346.935} C_VEL
LIN {X 0,Y 380.838,Z 249.278,A -85,B 0,C 180,E1 -12347.658,E2 -12347.658} C_VEL
LIN {X 0,Y 381.526,Z 238.634,A -85,B 0,C 180,E1 -12348.249,E2 -12348.249} C_VEL
LIN {X 0,Y 382.23,Z 225.355,A -85,B 0,C 180,E1 -12348.77,E2 -12348.77} C_VEL
LIN {X 0,Y 382.674,Z 207.053,A -85,B 0,C 180,E1 -12349.165,E2 -12349.165} C_VEL
LIN {X 0,Y 383.305,Z 146.764,A -85,B 0,C 180,E1 -12350.306,E2 -12350.306} C_VEL
LIN {X 0,Y 378.29,Z 119.671,A -85,B 0,C 180,E1 -12351.123,E2 -12351.123} C_VEL
LIN {X 0,Y 377.479,Z 115.277,A -85,B 0,C 180,E1 -12351.306,E2 -12351.306} C_VEL
LIN {X 0,Y 378.777,Z 101.452,A -85,B 0,C 180,E1 -12355.262,E2 -12355.262} C_VEL
LIN {X 0,Y 378.742,Z 97.44,A -85,B 0,C 180,E1 -12356.445,E2 -12356.445} C_VEL
LIN {X 0,Y 376.829,Z 87.129,A -85,B 0,C 180,E1 -12359.619,E2 -12359.619} C_VEL
LIN {X 0,Y 375.978,Z 83.184,A -85,B 0,C 180,E1 -12360.965,E2 -12360.965} C_VEL
LIN {X 0,Y 375.982,Z 83.142,A -85,B 0,C 180,E1 -12364.667,E2 -12364.667} C_VEL
LIN {X 0,Y 375.977,Z 83.148,A -85,B 0,C 180,E1 -12368.27,E2 -12368.27} C_VEL
LIN {X 0,Y 375.936,Z 83.145,A -85,B 0,C 180,E1 -12371.6,E2 -12371.6} C_VEL
LIN {X 0,Y 375.928,Z 83.152,A -85,B 0,C 180,E1 -12375.268,E2 -12375.268} C_VEL
LIN {X 0,Y 375.936,Z 83.154,A -85,B 0,C 180,E1 -12378.399,E2 -12378.399} C_VEL
LIN {X 0,Y 375.974,Z 83.152,A -85,B 0,C 180,E1 -12381.729,E2 -12381.729} C_VEL
LIN {X 0,Y 375.981,Z 83.135,A -85,B 0,C 180,E1 -12385.332,E2 -12385.332} C_VEL
LIN {X 0,Y 375.959,Z 83.151,A -85,B 0,C 180,E1 -12388.438,E2 -12388.438} C_VEL
LIN {X 0,Y 375.984,Z 83.136,A -85,B 0,C 180,E1 -12392.14,E2 -12392.14} C_VEL
LIN {X 0,Y 376.007,Z 83.134,A -85,B 0,C 180,E1 -12394.538,E2 -12394.538} C_VEL
LIN {X 0,Y 375.969,Z 83.149,A -85,B 0,C 180,E1 -12398.046,E2 -12398.046} C_VEL
LIN {X 0,Y 376.009,Z 83.121,A -85,B 0,C 180,E1 -12401.473,E2 -12401.473} C_VEL
LIN {X 0,Y 376.059,Z 83.14,A -85,B 0,C 180,E1 -12404.832,E2 -12404.832} C_VEL
LIN {X 0,Y 376.05,Z 83.13,A -85,B 0,C 180,E1 -12408.136,E2 -12408.136} C_VEL
LIN {X 0,Y 376.258,Z 83.097,A -85,B 0,C 180,E1 -12411.876,E2 -12411.876} C_VEL
LIN {X 0,Y 376.175,Z 83.126,A -85,B 0,C 180,E1 -12414.639,E2 -12414.639} C_VEL
LIN {X 0,Y 376.351,Z 83.093,A -85,B 0,C 180,E1 -12417.859,E2 -12417.859} C_VEL
LIN {X 0,Y 376.487,Z 83.06,A -85,B 0,C 180,E1 -12419.999,E2 -12419.999} C_VEL
LIN {X 0,Y 376.184,Z 83.118,A -85,B 0,C 180,E1 -12423.212,E2 -12423.212} C_VEL
LIN {X 0,Y 376.234,Z 83.112,A -85,B 0,C 180,E1 -12426.618,E2 -12426.618} C_VEL
LIN {X 0,Y 376.205,Z 83.104,A -85,B 0,C 180,E1 -12428.594,E2 -12428.594} C_VEL
LIN {X 0,Y 376.057,Z 83.13,A -85,B 0,C 180,E1 -12431.863,E2 -12431.863} C_VEL
LIN {X 0,Y 376.058,Z 83.143,A -85,B 0,C 180,E1 -12435.167,E2 -12435.167} C_VEL
LIN {X 0,Y 376.007,Z 83.126,A -85,B 0,C 180,E1 -12438.526,E2 -12438.526} C_VEL
LIN {X 0,Y 375.966,Z 83.15,A -85,B 0,C 180,E1 -12441.953,E2 -12441.953} C_VEL
LIN {X 0,Y 376.004,Z 83.138,A -85,B 0,C 180,E1 -12445.46,E2 -12445.46} C_VEL
LIN {X 0,Y 375.959,Z 83.146,A -85,B 0,C 180,E1 -12449.079,E2 -12449.079} C_VEL
LIN {X 0,Y 375.946,Z 83.149,A -85,B 0,C 180,E1 -12452.828,E2 -12452.828} C_VEL
LIN {X 0,Y 375.956,Z 83.146,A -85,B 0,C 180,E1 -12455.415,E2 -12455.415} C_VEL
LIN {X 0,Y 375.975,Z 83.153,A -85,B 0,C 180,E1 -12458.271,E2 -12458.271} C_VEL
LIN {X 0,Y 375.957,Z 83.147,A -85,B 0,C 180,E1 -12461.605,E2 -12461.605} C_VEL
LIN {X 0,Y 375.923,Z 83.148,A -85,B 0,C 180,E1 -12465.268,E2 -12465.268} C_VEL
LIN {X 0,Y 375.93,Z 83.119,A -85,B 0,C 180,E1 -12468.399,E2 -12468.399} C_VEL
LIN {X 0,Y 375.972,Z 83.152,A -85,B 0,C 180,E1 -12471.729,E2 -12471.729} C_VEL
LIN {X 0,Y 375.976,Z 83.125,A -85,B 0,C 180,E1 -12475.332,E2 -12475.332} C_VEL
LIN {X 0,Y 375.954,Z 83.155,A -85,B 0,C 180,E1 -12478.438,E2 -12478.438} C_VEL
LIN {X 0,Y 375.979,Z 83.147,A -85,B 0,C 180,E1 -12482.14,E2 -12482.14} C_VEL
LIN {X 0,Y 376.003,Z 83.149,A -85,B 0,C 180,E1 -12484.539,E2 -12484.539} C_VEL
LIN {X 0,Y 375.96,Z 83.157,A -85,B 0,C 180,E1 -12488.046,E2 -12488.046} C_VEL
LIN {X 0,Y 376.02,Z 83.149,A -85,B 0,C 180,E1 -12491.474,E2 -12491.474} C_VEL
LIN {X 0,Y 376.055,Z 83.144,A -85,B 0,C 180,E1 -12494.833,E2 -12494.833} C_VEL
LIN {X 0,Y 376.116,Z 83.431,A -85,B 0,C 180,E1 -12496.109,E2 -12496.109} C_VEL
LIN {X 0,Y 376.404,Z 84.52,A -85,B 0,C 180,E1 -12496.466,E2 -12496.466} C_VEL
LIN {X 0,Y 377.861,Z 87.022,A -85,B 0,C 180,E1 -12497.103,E2 -12497.103} C_VEL
LIN {X 0,Y 380.043,Z 88.683,A -85,B 0,C 180,E1 -12497.945,E2 -12497.945} C_VEL
LIN {X 0,Y 381.206,Z 89.429,A -85,B 0,C 180,E1 -12498.434,E2 -12498.434} C_VEL
LIN {X 0,Y 382.608,Z 91.818,A -85,B 0,C 180,E1 -12499.081,E2 -12499.081} C_VEL
LIN {X 0,Y 384.915,Z 94.149,A -85,B 0,C 180,E1 -12500.234,E2 -12500.234} C_VEL
LIN {X 0,Y 387.592,Z 95.673,A -85,B 0,C 180,E1 -12501.659,E2 -12501.659} C_VEL
LIN {X 0,Y 389.285,Z 98.435,A -85,B 0,C 180,E1 -12502.841,E2 -12502.841} C_VEL
LIN {X 0,Y 391.041,Z 100.14,A -85,B 0,C 180,E1 -12504.198,E2 -12504.198} C_VEL
LIN {X 0,Y 392.756,Z 101.219,A -85,B 0,C 180,E1 -12505.895,E2 -12505.895} C_VEL
LIN {X 0,Y 393.915,Z 101.599,A -85,B 0,C 180,E1 -12507.579,E2 -12507.579} C_VEL
LIN {X 0,Y 394.453,Z 102.033,A -85,B 0,C 180,E1 -12508.979,E2 -12508.979} C_VEL
LIN {X 0,Y 394.593,Z 101.943,A -85,B 0,C 180,E1 -12510,E2 -12510} C_VEL
LIN {X 0,Y 394.096,Z 101.716,A -85,B 0,C 180,E1 -12512.044,E2 -12512.044} C_VEL
LIN {X 0,Y 393.066,Z 101.32,A -85,B 0,C 180,E1 -12513.725,E2 -12513.725} C_VEL
LIN {X 0,Y 391.609,Z 100.582,A -85,B 0,C 180,E1 -12515.277,E2 -12515.277} C_VEL
LIN {X 0,Y 389.867,Z 99.109,A -85,B 0,C 180,E1 -12516.729,E2 -12516.729} C_VEL
LIN {X 0,Y 388.032,Z 96.481,A -85,B 0,C 180,E1 -12518.061,E2 -12518.061} C_VEL
LIN {X 0,Y 387.368,Z 95.385,A -85,B 0,C 180,E1 -12518.477,E2 -12518.477} C_VEL
LIN {X 0,Y 384.676,Z 93.969,A -85,B 0,C 180,E1 -12519.881,E2 -12519.881} C_VEL
LIN {X 0,Y 382.442,Z 91.628,A -85,B 0,C 180,E1 -12520.991,E2 -12520.991} C_VEL
LIN {X 0,Y 380.868,Z 89.114,A -85,B 0,C 180,E1 -12521.711,E2 -12521.711} C_VEL
LIN {X 0,Y 378.261,Z 87.428,A -85,B 0,C 180,E1 -12522.746,E2 -12522.746} C_VEL
LIN {X 0,Y 376.574,Z 84.984,A -85,B 0,C 180,E1 -12523.445,E2 -12523.445} C_VEL
LIN {X 0,Y 376.201,Z 83.746,A -85,B 0,C 180,E1 -12523.73,E2 -12523.73} C_VEL
LIN {X 0,Y 376.064,Z 83.165,A -85,B 0,C 180,E1 -12524.337,E2 -12524.337} C_VEL
LIN {X 0,Y 376.04,Z 83.146,A -85,B 0,C 180,E1 -12527.608,E2 -12527.608} C_VEL
LIN {X 0,Y 375.974,Z 83.154,A -85,B 0,C 180,E1 -12530.832,E2 -12530.832} C_VEL
LIN {X 0,Y 375.99,Z 83.152,A -85,B 0,C 180,E1 -12534.282,E2 -12534.282} C_VEL
LIN {X 0,Y 376.016,Z 83.148,A -85,B 0,C 180,E1 -12536.652,E2 -12536.652} C_VEL
LIN {X 0,Y 375.961,Z 83.142,A -85,B 0,C 180,E1 -12540.313,E2 -12540.313} C_VEL
LIN {X 0,Y 375.956,Z 83.127,A -85,B 0,C 180,E1 -12544.112,E2 -12544.112} C_VEL
LIN {X 0,Y 375.951,Z 83.151,A -85,B 0,C 180,E1 -12546.741,E2 -12546.741} C_VEL
LIN {X 0,Y 375.98,Z 83.135,A -85,B 0,C 180,E1 -12550.026,E2 -12550.026} C_VEL
LIN {X 0,Y 375.246,Z 83.213,A -85,B 0,C 180,E1 -12550.919,E2 -12550.919} C_VEL
LIN {X 0,Y 372.338,Z 83.565,A -85,B 0,C 180,E1 -12552.371,E2 -12552.371} C_VEL
LIN {X 0,Y 369.933,Z 83.875,A -85,B 0,C 180,E1 -12553.546,E2 -12553.546} C_VEL
LIN {X 0,Y 368.937,Z 84.017,A -85,B 0,C 180,E1 -12554.454,E2 -12554.454} C_VEL
LIN {X 0,Y 368.872,Z 84.025,A -85,B 0,C 180,E1 -12554.762,E2 -12554.762} C_VEL
LIN {X 0,Y 368.907,Z 84.025,A -85,B 0,C 180,E1 -12558.182,E2 -12558.182} C_VEL
LIN {X 0,Y 368.91,Z 84.032,A -85,B 0,C 180,E1 -12561.359,E2 -12561.359} C_VEL
LIN {X 0,Y 368.934,Z 84.015,A -85,B 0,C 180,E1 -12565.147,E2 -12565.147} C_VEL
LIN {X 0,Y 368.926,Z 84.034,A -85,B 0,C 180,E1 -12569.047,E2 -12569.047} C_VEL
LIN {X 0,Y 368.961,Z 84.006,A -85,B 0,C 180,E1 -12572.797,E2 -12572.797} C_VEL
LIN {X 0,Y 368.943,Z 84.025,A -85,B 0,C 180,E1 -12576.113,E2 -12576.113} C_VEL
LIN {X 0,Y 368.935,Z 84.012,A -85,B 0,C 180,E1 -12579.948,E2 -12579.948} C_VEL
LIN {X 0,Y 368.975,Z 84.017,A -85,B 0,C 180,E1 -12583.399,E2 -12583.399} C_VEL
LIN {X 0,Y 369.059,Z 84.009,A -85,B 0,C 180,E1 -12586.791,E2 -12586.791} C_VEL
LIN {X 0,Y 369.069,Z 83.985,A -85,B 0,C 180,E1 -12590.132,E2 -12590.132} C_VEL
LIN {X 0,Y 369.187,Z 83.984,A -85,B 0,C 180,E1 -12592.343,E2 -12592.343} C_VEL
LIN {X 0,Y 369.144,Z 84.003,A -85,B 0,C 180,E1 -12594.538,E2 -12594.538} C_VEL
LIN {X 0,Y 369.316,Z 83.968,A -85,B 0,C 180,E1 -12597.819,E2 -12597.819} C_VEL
LIN {X 0,Y 369.456,Z 83.935,A -85,B 0,C 180,E1 -12600.001,E2 -12600.001} C_VEL
LIN {X 0,Y 369.316,Z 83.97,A -85,B 0,C 180,E1 -12602.182,E2 -12602.182} C_VEL
LIN {X 0,Y 369.213,Z 83.987,A -85,B 0,C 180,E1 -12606.559,E2 -12606.559} C_VEL
LIN {X 0,Y 369.138,Z 83.981,A -85,B 0,C 180,E1 -12608.761,E2 -12608.761} C_VEL
LIN {X 0,Y 369.006,Z 84.011,A -85,B 0,C 180,E1 -12612.094,E2 -12612.094} C_VEL
LIN {X 0,Y 368.998,Z 84.018,A -85,B 0,C 180,E1 -12615.465,E2 -12615.465} C_VEL
LIN {X 0,Y 368.959,Z 83.998,A -85,B 0,C 180,E1 -12618.895,E2 -12618.895} C_VEL
LIN {X 0,Y 368.936,Z 84.024,A -85,B 0,C 180,E1 -12622.395,E2 -12622.395} C_VEL
LIN {X 0,Y 369.001,Z 84.003,A -85,B 0,C 180,E1 -12625.981,E2 -12625.981} C_VEL
LIN {X 0,Y 368.916,Z 84.029,A -85,B 0,C 180,E1 -12629.691,E2 -12629.691} C_VEL
LIN {X 0,Y 368.898,Z 84.021,A -85,B 0,C 180,E1 -12633.044,E2 -12633.044} C_VEL
LIN {X 0,Y 368.918,Z 84.025,A -85,B 0,C 180,E1 -12636.197,E2 -12636.197} C_VEL
LIN {X 0,Y 368.903,Z 84.026,A -85,B 0,C 180,E1 -12638.954,E2 -12638.954} C_VEL
LIN {X 0,Y 368.883,Z 84.033,A -85,B 0,C 180,E1 -12642.01,E2 -12642.01} C_VEL
LIN {X 0,Y 368.881,Z 84.03,A -85,B 0,C 180,E1 -12645.176,E2 -12645.176} C_VEL
LIN {X 0,Y 368.885,Z 84.026,A -85,B 0,C 180,E1 -12648.178,E2 -12648.178} C_VEL
LIN {X 0,Y 368.911,Z 84.024,A -85,B 0,C 180,E1 -12651.36,E2 -12651.36} C_VEL
LIN {X 0,Y 368.939,Z 84.016,A -85,B 0,C 180,E1 -12655.147,E2 -12655.147} C_VEL
LIN {X 0,Y 368.96,Z 84.229,A -85,B 0,C 180,E1 -12658.819,E2 -12658.819} C_VEL
LIN {X 0,Y 370.708,Z 92.802,A -85,B 0,C 180,E1 -12661.709,E2 -12661.709} C_VEL
LIN {X 0,Y 371.876,Z 100.113,A -85,B 0,C 180,E1 -12663.935,E2 -12663.935} C_VEL
LIN {X 0,Y 371.345,Z 107.213,A -85,B 0,C 180,E1 -12665.99,E2 -12665.99} C_VEL
LIN {X 0,Y 370.553,Z 115.052,A -85,B 0,C 180,E1 -12668.267,E2 -12668.267} C_VEL
LIN {X 0,Y 371.471,Z 119.73,A -85,B 0,C 180,E1 -12668.475,E2 -12668.475} C_VEL
LIN {X 0,Y 376.629,Z 147.632,A -85,B 0,C 180,E1 -12669.339,E2 -12669.339} C_VEL
LIN {X 0,Y 375.692,Z 219.861,A -85,B 0,C 180,E1 -12670.749,E2 -12670.749} C_VEL
LIN {X 0,Y 375.289,Z 229.757,A -85,B 0,C 180,E1 -12671.047,E2 -12671.047} C_VEL
LIN {X 0,Y 374.665,Z 239.73,A -85,B 0,C 180,E1 -12671.475,E2 -12671.475} C_VEL
LIN {X 0,Y 374.058,Z 249.087,A -85,B 0,C 180,E1 -12672.011,E2 -12672.011} C_VEL
LIN {X 0,Y 373.169,Z 259.226,A -85,B 0,C 180,E1 -12672.745,E2 -12672.745} C_VEL
LIN {X 0,Y 372.368,Z 268.223,A -85,B 0,C 180,E1 -12673.554,E2 -12673.554} C_VEL
LIN {X 0,Y 371.474,Z 276.95,A -85,B 0,C 180,E1 -12674.5,E2 -12674.5} C_VEL
LIN {X 0,Y 370.715,Z 284.75,A -85,B 0,C 180,E1 -12675.511,E2 -12675.511} C_VEL
LIN {X 0,Y 369.886,Z 293.194,A -85,B 0,C 180,E1 -12676.82,E2 -12676.82} C_VEL
LIN {X 0,Y 369.243,Z 299.144,A -85,B 0,C 180,E1 -12677.915,E2 -12677.915} C_VEL
LIN {X 0,Y 368.561,Z 305.46,A -85,B 0,C 180,E1 -12679.285,E2 -12679.285} C_VEL
LIN {X 0,Y 368.106,Z 310.722,A -85,B 0,C 180,E1 -12680.66,E2 -12680.66} C_VEL
LIN {X 0,Y 367.718,Z 315.852,A -85,B 0,C 180,E1 -12682.312,E2 -12682.312} C_VEL
LIN {X 0,Y 367.504,Z 319.818,A -85,B 0,C 180,E1 -12683.953,E2 -12683.953} C_VEL
LIN {X 0,Y 367.437,Z 322.789,A -85,B 0,C 180,E1 -12685.612,E2 -12685.612} C_VEL
LIN {X 0,Y 367.36,Z 325.233,A -85,B 0,C 180,E1 -12687.807,E2 -12687.807} C_VEL
LIN {X 0,Y 367.404,Z 325.823,A -85,B 0,C 180,E1 -12688.904,E2 -12688.904} C_VEL
LIN {X 0,Y 367.404,Z 325.823,A -85,B 0,C 180,E1 -12691.096,E2 -12691.096} C_VEL
LIN {X 0,Y 367.36,Z 325.233,A -85,B 0,C 180,E1 -12692.193,E2 -12692.193} C_VEL
LIN {X 0,Y 367.436,Z 322.789,A -85,B 0,C 180,E1 -12694.388,E2 -12694.388} C_VEL
LIN {X 0,Y 367.479,Z 319.899,A -85,B 0,C 180,E1 -12696.011,E2 -12696.011} C_VEL
LIN {X 0,Y 367.718,Z 315.852,A -85,B 0,C 180,E1 -12697.688,E2 -12697.688} C_VEL
LIN {X 0,Y 368.106,Z 310.722,A -85,B 0,C 180,E1 -12699.34,E2 -12699.34} C_VEL
LIN {X 0,Y 368.561,Z 305.46,A -85,B 0,C 180,E1 -12700.715,E2 -12700.715} C_VEL
LIN {X 0,Y 369.242,Z 299.144,A -85,B 0,C 180,E1 -12702.085,E2 -12702.085} C_VEL
LIN {X 0,Y 369.874,Z 293.193,A -85,B 0,C 180,E1 -12703.18,E2 -12703.18} C_VEL
LIN {X 0,Y 370.576,Z 286.266,A -85,B 0,C 180,E1 -12704.273,E2 -12704.273} C_VEL
LIN {X 0,Y 371.392,Z 278.085,A -85,B 0,C 180,E1 -12705.363,E2 -12705.363} C_VEL
LIN {X 0,Y 372.199,Z 269.573,A -85,B 0,C 180,E1 -12706.312,E2 -12706.312} C_VEL
LIN {X 0,Y 373.038,Z 260.858,A -85,B 0,C 180,E1 -12707.12,E2 -12707.12} C_VEL
LIN {X 0,Y 373.863,Z 251.1,A -85,B 0,C 180,E1 -12707.857,E2 -12707.857} C_VEL
LIN {X 0,Y 374.497,Z 242.306,A -85,B 0,C 180,E1 -12708.392,E2 -12708.392} C_VEL
LIN {X 0,Y 375.143,Z 232.379,A -85,B 0,C 180,E1 -12708.854,E2 -12708.854} C_VEL
LIN {X 0,Y 375.581,Z 222.523,A -85,B 0,C 180,E1 -12709.186,E2 -12709.186} C_VEL
LIN {X 0,Y 376.088,Z 199.703,A -85,B 0,C 180,E1 -12709.656,E2 -12709.656} C_VEL
LIN {X 0,Y 376.716,Z 148.141,A -85,B 0,C 180,E1 -12710.646,E2 -12710.646} C_VEL
LIN {X 0,Y 371.67,Z 120.741,A -85,B 0,C 180,E1 -12711.492,E2 -12711.492} C_VEL
LIN {X 0,Y 370.538,Z 115.234,A -85,B 0,C 180,E1 -12711.709,E2 -12711.709} C_VEL
LIN {X 0,Y 370.662,Z 113.023,A -85,B 0,C 180,E1 -12712.285,E2 -12712.285} C_VEL
LIN {X 0,Y 371.771,Z 103.163,A -85,B 0,C 180,E1 -12715.205,E2 -12715.205} C_VEL
LIN {X 0,Y 371.847,Z 99.263,A -85,B 0,C 180,E1 -12716.369,E2 -12716.369} C_VEL
LIN {X 0,Y 370.229,Z 90.376,A -85,B 0,C 180,E1 -12719.165,E2 -12719.165} C_VEL
LIN {X 0,Y 368.947,Z 84.09,A -85,B 0,C 180,E1 -12721.27,E2 -12721.27} C_VEL
LIN {X 0,Y 368.932,Z 84.017,A -85,B 0,C 180,E1 -12725.001,E2 -12725.001} C_VEL
LIN {X 0,Y 368.911,Z 84.024,A -85,B 0,C 180,E1 -12728.64,E2 -12728.64} C_VEL
LIN {X 0,Y 368.883,Z 84.03,A -85,B 0,C 180,E1 -12732.009,E2 -12732.009} C_VEL
LIN {X 0,Y 368.881,Z 84.03,A -85,B 0,C 180,E1 -12735.175,E2 -12735.175} C_VEL
LIN {X 0,Y 368.884,Z 84.033,A -85,B 0,C 180,E1 -12738.177,E2 -12738.177} C_VEL
LIN {X 0,Y 368.908,Z 84.029,A -85,B 0,C 180,E1 -12741.36,E2 -12741.36} C_VEL
LIN {X 0,Y 368.938,Z 84.013,A -85,B 0,C 180,E1 -12745.146,E2 -12745.146} C_VEL
LIN {X 0,Y 368.93,Z 84.032,A -85,B 0,C 180,E1 -12749.046,E2 -12749.046} C_VEL
LIN {X 0,Y 368.964,Z 84.005,A -85,B 0,C 180,E1 -12752.796,E2 -12752.796} C_VEL
LIN {X 0,Y 368.946,Z 84.023,A -85,B 0,C 180,E1 -12756.112,E2 -12756.112} C_VEL
LIN {X 0,Y 368.938,Z 84.012,A -85,B 0,C 180,E1 -12759.947,E2 -12759.947} C_VEL
LIN {X 0,Y 368.977,Z 84.013,A -85,B 0,C 180,E1 -12763.398,E2 -12763.398} C_VEL
LIN {X 0,Y 369.058,Z 84.007,A -85,B 0,C 180,E1 -12766.79,E2 -12766.79} C_VEL
LIN {X 0,Y 369.068,Z 83.984,A -85,B 0,C 180,E1 -12770.131,E2 -12770.131} C_VEL
LIN {X 0,Y 369.189,Z 83.983,A -85,B 0,C 180,E1 -12772.342,E2 -12772.342} C_VEL
LIN {X 0,Y 369.148,Z 84.002,A -85,B 0,C 180,E1 -12774.537,E2 -12774.537} C_VEL
LIN {X 0,Y 369.316,Z 83.97,A -85,B 0,C 180,E1 -12777.818,E2 -12777.818} C_VEL
LIN {X 0,Y 369.456,Z 83.935,A -85,B 0,C 180,E1 -12779.999,E2 -12779.999} C_VEL
LIN {X 0,Y 369.316,Z 83.968,A -85,B 0,C 180,E1 -12782.181,E2 -12782.181} C_VEL
LIN {X 0,Y 369.204,Z 83.988,A -85,B 0,C 180,E1 -12786.605,E2 -12786.605} C_VEL
LIN {X 0,Y 369.137,Z 83.984,A -85,B 0,C 180,E1 -12788.76,E2 -12788.76} C_VEL
LIN {X 0,Y 369.012,Z 84.011,A -85,B 0,C 180,E1 -12792.092,E2 -12792.092} C_VEL
LIN {X 0,Y 368.997,Z 84.02,A -85,B 0,C 180,E1 -12795.464,E2 -12795.464} C_VEL
LIN {X 0,Y 368.956,Z 84.002,A -85,B 0,C 180,E1 -12798.894,E2 -12798.894} C_VEL
LIN {X 0,Y 368.934,Z 84.025,A -85,B 0,C 180,E1 -12802.394,E2 -12802.394} C_VEL
LIN {X 0,Y 368.998,Z 84.008,A -85,B 0,C 180,E1 -12805.98,E2 -12805.98} C_VEL
LIN {X 0,Y 368.912,Z 84.029,A -85,B 0,C 180,E1 -12809.69,E2 -12809.69} C_VEL
LIN {X 0,Y 368.894,Z 84.025,A -85,B 0,C 180,E1 -12813.043,E2 -12813.043} C_VEL
LIN {X 0,Y 368.916,Z 84.025,A -85,B 0,C 180,E1 -12816.196,E2 -12816.196} C_VEL
LIN {X 0,Y 368.905,Z 84.028,A -85,B 0,C 180,E1 -12818.952,E2 -12818.952} C_VEL
LIN {X 0,Y 368.906,Z 84.026,A -85,B 0,C 180,E1 -12822.014,E2 -12822.014} C_VEL
LIN {X 0,Y 368.876,Z 84.026,A -85,B 0,C 180,E1 -12825.175,E2 -12825.175} C_VEL
LIN {X 0,Y 368.878,Z 83.995,A -85,B 0,C 180,E1 -12828.177,E2 -12828.177} C_VEL
LIN {X 0,Y 368.907,Z 84.031,A -85,B 0,C 180,E1 -12831.359,E2 -12831.359} C_VEL
LIN {X 0,Y 368.933,Z 84.002,A -85,B 0,C 180,E1 -12835.146,E2 -12835.146} C_VEL
LIN {X 0,Y 368.925,Z 84.028,A -85,B 0,C 180,E1 -12839.046,E2 -12839.046} C_VEL
LIN {X 0,Y 368.959,Z 84.027,A -85,B 0,C 180,E1 -12842.796,E2 -12842.796} C_VEL
LIN {X 0,Y 368.942,Z 84.031,A -85,B 0,C 180,E1 -12846.113,E2 -12846.113} C_VEL
LIN {X 0,Y 368.933,Z 84.031,A -85,B 0,C 180,E1 -12849.947,E2 -12849.947} C_VEL
LIN {X 0,Y 368.973,Z 84.026,A -85,B 0,C 180,E1 -12853.399,E2 -12853.399} C_VEL
LIN {X 0,Y 369.037,Z 84.421,A -85,B 0,C 180,E1 -12854.112,E2 -12854.112} C_VEL
LIN {X 0,Y 369.449,Z 85.783,A -85,B 0,C 180,E1 -12854.431,E2 -12854.431} C_VEL
LIN {X 0,Y 370.843,Z 87.963,A -85,B 0,C 180,E1 -12854.93,E2 -12854.93} C_VEL
LIN {X 0,Y 373.911,Z 90.221,A -85,B 0,C 180,E1 -12855.939,E2 -12855.939} C_VEL
LIN {X 0,Y 375.803,Z 93.292,A -85,B 0,C 180,E1 -12856.694,E2 -12856.694} C_VEL
LIN {X 0,Y 378.432,Z 95.423,A -85,B 0,C 180,E1 -12857.668,E2 -12857.668} C_VEL
LIN {X 0,Y 379.53,Z 96.232,A -85,B 0,C 180,E1 -12858.131,E2 -12858.131} C_VEL
LIN {X 0,Y 381.567,Z 99.132,A -85,B 0,C 180,E1 -12859.051,E2 -12859.051} C_VEL
LIN {X 0,Y 384.055,Z 101.302,A -85,B 0,C 180,E1 -12860.262,E2 -12860.262} C_VEL
LIN {X 0,Y 386.289,Z 102.545,A -85,B 0,C 180,E1 -12861.433,E2 -12861.433} C_VEL
LIN {X 0,Y 388.224,Z 105.441,A -85,B 0,C 180,E1 -12862.72,E2 -12862.72} C_VEL
LIN {X 0,Y 390.287,Z 107.323,A -85,B 0,C 180,E1 -12864.316,E2 -12864.316} C_VEL
LIN {X 0,Y 391.884,Z 108.243,A -85,B 0,C 180,E1 -12865.886,E2 -12865.886} C_VEL
LIN {X 0,Y 392.994,Z 108.615,A -85,B 0,C 180,E1 -12867.456,E2 -12867.456} C_VEL
LIN {X 0,Y 393.615,Z 109.062,A -85,B 0,C 180,E1 -12869.07,E2 -12869.07} C_VEL
LIN {X 0,Y 393.595,Z 109.005,A -85,B 0,C 180,E1 -12870.729,E2 -12870.729} C_VEL
LIN {X 0,Y 393.23,Z 108.759,A -85,B 0,C 180,E1 -12872.048,E2 -12872.048} C_VEL
LIN {X 0,Y 392.191,Z 108.365,A -85,B 0,C 180,E1 -12873.733,E2 -12873.733} C_VEL
LIN {X 0,Y 390.718,Z 107.632,A -85,B 0,C 180,E1 -12875.289,E2 -12875.289} C_VEL
LIN {X 0,Y 388.952,Z 106.205,A -85,B 0,C 180,E1 -12876.745,E2 -12876.745} C_VEL
LIN {X 0,Y 387.179,Z 103.953,A -85,B 0,C 180,E1 -12878.011,E2 -12878.011} C_VEL
LIN {X 0,Y 385.95,Z 102.185,A -85,B 0,C 180,E1 -12878.772,E2 -12878.772} C_VEL
LIN {X 0,Y 383.231,Z 100.733,A -85,B 0,C 180,E1 -12880.134,E2 -12880.134} C_VEL
LIN {X 0,Y 380.895,Z 98.355,A -85,B 0,C 180,E1 -12881.238,E2 -12881.238} C_VEL
LIN {X 0,Y 379.162,Z 95.784,A -85,B 0,C 180,E1 -12882.036,E2 -12882.036} C_VEL
LIN {X 0,Y 376.571,Z 94.099,A -85,B 0,C 180,E1 -12883.011,E2 -12883.011} C_VEL
LIN {X 0,Y 374.518,Z 91.35,A -85,B 0,C 180,E1 -12883.833,E2 -12883.833} C_VEL
LIN {X 0,Y 373.644,Z 89.87,A -85,B 0,C 180,E1 -12884.154,E2 -12884.154} C_VEL
LIN {X 0,Y 370.852,Z 87.966,A -85,B 0,C 180,E1 -12885.068,E2 -12885.068} C_VEL
LIN {X 0,Y 369.45,Z 85.786,A -85,B 0,C 180,E1 -12885.569,E2 -12885.569} C_VEL
LIN {X 0,Y 369.037,Z 84.424,A -85,B 0,C 180,E1 -12885.888,E2 -12885.888} C_VEL
LIN {X 0,Y 368.973,Z 84.026,A -85,B 0,C 180,E1 -12886.601,E2 -12886.601} C_VEL
LIN {X 0,Y 368.933,Z 84.032,A -85,B 0,C 180,E1 -12890.053,E2 -12890.053} C_VEL
LIN {X 0,Y 368.942,Z 84.031,A -85,B 0,C 180,E1 -12893.887,E2 -12893.887} C_VEL
LIN {X 0,Y 368.959,Z 84.027,A -85,B 0,C 180,E1 -12897.204,E2 -12897.204} C_VEL
LIN {X 0,Y 368.925,Z 84.028,A -85,B 0,C 180,E1 -12900.954,E2 -12900.954} C_VEL
LIN {X 0,Y 368.926,Z 84,A -85,B 0,C 180,E1 -12905.002,E2 -12905.002} C_VEL
LIN {X 0,Y 368.907,Z 84.031,A -85,B 0,C 180,E1 -12908.641,E2 -12908.641} C_VEL
LIN {X 0,Y 368.877,Z 83.995,A -85,B 0,C 180,E1 -12912.01,E2 -12912.01} C_VEL
LIN {X 0,Y 368.872,Z 84.025,A -85,B 0,C 180,E1 -12914.762,E2 -12914.762} C_VEL
LIN {X 0,Y 368.25,Z 84.116,A -85,B 0,C 180,E1 -12915.673,E2 -12915.673} C_VEL
LIN {X 0,Y 365.413,Z 84.469,A -85,B 0,C 180,E1 -12917.155,E2 -12917.155} C_VEL
LIN {X 0,Y 362.985,Z 84.762,A -85,B 0,C 180,E1 -12918.354,E2 -12918.354} C_VEL
LIN {X 0,Y 361.944,Z 84.888,A -85,B 0,C 180,E1 -12919.281,E2 -12919.281} C_VEL
LIN {X 0,Y 361.862,Z 84.898,A -85,B 0,C 180,E1 -12919.595,E2 -12919.595} C_VEL
LIN {X 0,Y 361.867,Z 84.912,A -85,B 0,C 180,E1 -12922.983,E2 -12922.983} C_VEL
LIN {X 0,Y 361.856,Z 84.898,A -85,B 0,C 180,E1 -12926.631,E2 -12926.631} C_VEL
LIN {X 0,Y 361.87,Z 84.907,A -85,B 0,C 180,E1 -12929.672,E2 -12929.672} C_VEL
LIN {X 0,Y 361.952,Z 84.882,A -85,B 0,C 180,E1 -12933.476,E2 -12933.476} C_VEL
LIN {X 0,Y 361.89,Z 84.905,A -85,B 0,C 180,E1 -12937.145,E2 -12937.145} C_VEL
LIN {X 0,Y 361.905,Z 84.879,A -85,B 0,C 180,E1 -12940.724,E2 -12940.724} C_VEL
LIN {X 0,Y 361.932,Z 84.893,A -85,B 0,C 180,E1 -12943.067,E2 -12943.067} C_VEL
LIN {X 0,Y 361.999,Z 84.891,A -85,B 0,C 180,E1 -12946.528,E2 -12946.528} C_VEL
LIN {X 0,Y 362.033,Z 84.86,A -85,B 0,C 180,E1 -12949.939,E2 -12949.939} C_VEL
LIN {X 0,Y 362.15,Z 84.859,A -85,B 0,C 180,E1 -12952.193,E2 -12952.193} C_VEL
LIN {X 0,Y 362.117,Z 84.88,A -85,B 0,C 180,E1 -12954.432,E2 -12954.432} C_VEL
LIN {X 0,Y 362.28,Z 84.845,A -85,B 0,C 180,E1 -12957.777,E2 -12957.777} C_VEL
LIN {X 0,Y 362.426,Z 84.81,A -85,B 0,C 180,E1 -12960.001,E2 -12960.001} C_VEL
LIN {X 0,Y 362.28,Z 84.846,A -85,B 0,C 180,E1 -12962.224,E2 -12962.224} C_VEL
LIN {X 0,Y 362.176,Z 84.863,A -85,B 0,C 180,E1 -12966.687,E2 -12966.687} C_VEL
LIN {X 0,Y 362.074,Z 84.858,A -85,B 0,C 180,E1 -12968.934,E2 -12968.934} C_VEL
LIN {X 0,Y 361.961,Z 84.89,A -85,B 0,C 180,E1 -12972.333,E2 -12972.333} C_VEL
LIN {X 0,Y 361.962,Z 84.893,A -85,B 0,C 180,E1 -12974.621,E2 -12974.621} C_VEL
LIN {X 0,Y 361.957,Z 84.871,A -85,B 0,C 180,E1 -12978.1,E2 -12978.1} C_VEL
LIN {X 0,Y 361.894,Z 84.902,A -85,B 0,C 180,E1 -12981.653,E2 -12981.653} C_VEL
LIN {X 0,Y 361.929,Z 84.889,A -85,B 0,C 180,E1 -12985.291,E2 -12985.291} C_VEL
LIN {X 0,Y 361.909,Z 84.887,A -85,B 0,C 180,E1 -12987.78,E2 -12987.78} C_VEL
LIN {X 0,Y 361.838,Z 84.91,A -85,B 0,C 180,E1 -12991.63,E2 -12991.63} C_VEL
LIN {X 0,Y 361.875,Z 84.898,A -85,B 0,C 180,E1 -12995.345,E2 -12995.345} C_VEL
LIN {X 0,Y 361.87,Z 84.901,A -85,B 0,C 180,E1 -12999.027,E2 -12999.027} C_VEL
LIN {X 0,Y 361.838,Z 84.914,A -85,B 0,C 180,E1 -13002.829,E2 -13002.829} C_VEL
LIN {X 0,Y 361.82,Z 84.912,A -85,B 0,C 180,E1 -13005.947,E2 -13005.947} C_VEL
LIN {X 0,Y 361.837,Z 84.891,A -85,B 0,C 180,E1 -13009.245,E2 -13009.245} C_VEL
LIN {X 0,Y 361.873,Z 84.908,A -85,B 0,C 180,E1 -13012.776,E2 -13012.776} C_VEL
LIN {X 0,Y 361.857,Z 84.904,A -85,B 0,C 180,E1 -13015.72,E2 -13015.72} C_VEL
LIN {X 0,Y 361.913,Z 84.932,A -85,B 0,C 180,E1 -13018.378,E2 -13018.378} C_VEL
LIN {X 0,Y 363.462,Z 92.621,A -85,B 0,C 180,E1 -13021.092,E2 -13021.092} C_VEL
LIN {X 0,Y 364.893,Z 100.982,A -85,B 0,C 180,E1 -13023.705,E2 -13023.705} C_VEL
LIN {X 0,Y 364.714,Z 105.07,A -85,B 0,C 180,E1 -13024.917,E2 -13024.917} C_VEL
LIN {X 0,Y 363.649,Z 114.801,A -85,B 0,C 180,E1 -13027.822,E2 -13027.822} C_VEL
LIN {X 0,Y 364.072,Z 117.118,A -85,B 0,C 180,E1 -13027.965,E2 -13027.965} C_VEL
LIN {X 0,Y 369.362,Z 144.392,A -85,B 0,C 180,E1 -13028.851,E2 -13028.851} C_VEL
LIN {X 0,Y 370.106,Z 150.984,A -85,B 0,C 180,E1 -13029.029,E2 -13029.029} C_VEL
LIN {X 0,Y 369.008,Z 219.677,A -85,B 0,C 180,E1 -13030.386,E2 -13030.386} C_VEL
LIN {X 0,Y 368.532,Z 230.44,A -85,B 0,C 180,E1 -13030.722,E2 -13030.722} C_VEL
LIN {X 0,Y 367.932,Z 239.54,A -85,B 0,C 180,E1 -13031.124,E2 -13031.124} C_VEL
LIN {X 0,Y 367.208,Z 249.903,A -85,B 0,C 180,E1 -13031.736,E2 -13031.736} C_VEL
LIN {X 0,Y 366.395,Z 259.035,A -85,B 0,C 180,E1 -13032.416,E2 -13032.416} C_VEL
LIN {X 0,Y 365.558,Z 268.032,A -85,B 0,C 180,E1 -13033.239,E2 -13033.239} C_VEL
LIN {X 0,Y 364.606,Z 276.759,A -85,B 0,C 180,E1 -13034.201,E2 -13034.201} C_VEL
LIN {X 0,Y 363.779,Z 284.941,A -85,B 0,C 180,E1 -13035.285,E2 -13035.285} C_VEL
LIN {X 0,Y 362.934,Z 293.002,A -85,B 0,C 180,E1 -13036.563,E2 -13036.563} C_VEL
LIN {X 0,Y 362.268,Z 298.953,A -85,B 0,C 180,E1 -13037.678,E2 -13037.678} C_VEL
LIN {X 0,Y 361.546,Z 305.268,A -85,B 0,C 180,E1 -13039.075,E2 -13039.075} C_VEL
LIN {X 0,Y 361.058,Z 310.531,A -85,B 0,C 180,E1 -13040.477,E2 -13040.477} C_VEL
LIN {X 0,Y 360.668,Z 315.661,A -85,B 0,C 180,E1 -13042.16,E2 -13042.16} C_VEL
LIN {X 0,Y 360.499,Z 318.432,A -85,B 0,C 180,E1 -13043.283,E2 -13043.283} C_VEL
LIN {X 0,Y 360.385,Z 320.799,A -85,B 0,C 180,E1 -13044.404,E2 -13044.404} C_VEL
LIN {X 0,Y 360.348,Z 322.599,A -85,B 0,C 180,E1 -13045.526,E2 -13045.526} C_VEL
LIN {X 0,Y 360.264,Z 325.043,A -85,B 0,C 180,E1 -13047.764,E2 -13047.764} C_VEL
LIN {X 0,Y 360.304,Z 325.632,A -85,B 0,C 180,E1 -13048.882,E2 -13048.882} C_VEL
LIN {X 0,Y 360.361,Z 325.788,A -85,B 0,C 180,E1 -13050,E2 -13050} C_VEL
LIN {X 0,Y 360.304,Z 325.632,A -85,B 0,C 180,E1 -13051.118,E2 -13051.118} C_VEL
LIN {X 0,Y 360.264,Z 325.043,A -85,B 0,C 180,E1 -13052.236,E2 -13052.236} C_VEL
LIN {X 0,Y 360.348,Z 322.599,A -85,B 0,C 180,E1 -13054.474,E2 -13054.474} C_VEL
LIN {X 0,Y 360.379,Z 320.073,A -85,B 0,C 180,E1 -13055.961,E2 -13055.961} C_VEL
LIN {X 0,Y 360.591,Z 317.192,A -85,B 0,C 180,E1 -13057.278,E2 -13057.278} C_VEL
LIN {X 0,Y 360.918,Z 312.447,A -85,B 0,C 180,E1 -13058.962,E2 -13058.962} C_VEL
LIN {X 0,Y 361.467,Z 306.425,A -85,B 0,C 180,E1 -13060.644,E2 -13060.644} C_VEL
LIN {X 0,Y 362.095,Z 300.328,A -85,B 0,C 180,E1 -13062.043,E2 -13062.043} C_VEL
LIN {X 0,Y 362.763,Z 294.629,A -85,B 0,C 180,E1 -13063.158,E2 -13063.158} C_VEL
LIN {X 0,Y 363.688,Z 286.075,A -85,B 0,C 180,E1 -13064.549,E2 -13064.549} C_VEL
LIN {X 0,Y 364.526,Z 277.894,A -85,B 0,C 180,E1 -13065.659,E2 -13065.659} C_VEL
LIN {X 0,Y 365.373,Z 269.382,A -85,B 0,C 180,E1 -13066.626,E2 -13066.626} C_VEL
LIN {X 0,Y 366.248,Z 260.667,A -85,B 0,C 180,E1 -13067.447,E2 -13067.447} C_VEL
LIN {X 0,Y 367.117,Z 250.909,A -85,B 0,C 180,E1 -13068.197,E2 -13068.197} C_VEL
LIN {X 0,Y 367.756,Z 242.115,A -85,B 0,C 180,E1 -13068.741,E2 -13068.741} C_VEL
LIN {X 0,Y 368.444,Z 232.189,A -85,B 0,C 180,E1 -13069.21,E2 -13069.21} C_VEL
LIN {X 0,Y 368.888,Z 222.333,A -85,B 0,C 180,E1 -13069.548,E2 -13069.548} C_VEL
LIN {X 0,Y 369.409,Z 198.285,A -85,B 0,C 180,E1 -13070.051,E2 -13070.051} C_VEL
LIN {X 0,Y 370.01,Z 148.632,A -85,B 0,C 180,E1 -13071.024,E2 -13071.024} C_VEL
LIN {X 0,Y 365.086,Z 121.933,A -85,B 0,C 180,E1 -13071.871,E2 -13071.871} C_VEL
LIN {X 0,Y 363.638,Z 115.106,A -85,B 0,C 180,E1 -13072.136,E2 -13072.136} C_VEL
LIN {X 0,Y 363.79,Z 112.833,A -85,B 0,C 180,E1 -13072.729,E2 -13072.729} C_VEL
LIN {X 0,Y 364.901,Z 103.091,A -85,B 0,C 180,E1 -13075.68,E2 -13075.68} C_VEL
LIN {X 0,Y 364.704,Z 99.226,A -85,B 0,C 180,E1 -13076.88,E2 -13076.88} C_VEL
LIN {X 0,Y 363.007,Z 90.319,A -85,B 0,C 180,E1 -13079.766,E2 -13079.766} C_VEL
LIN {X 0,Y 361.913,Z 84.94,A -85,B 0,C 180,E1 -13081.622,E2 -13081.622} C_VEL
LIN {X 0,Y 361.871,Z 84.895,A -85,B 0,C 180,E1 -13085.636,E2 -13085.636} C_VEL
LIN {X 0,Y 361.872,Z 84.893,A -85,B 0,C 180,E1 -13089.026,E2 -13089.026} C_VEL
LIN {X 0,Y 361.838,Z 84.912,A -85,B 0,C 180,E1 -13092.828,E2 -13092.828} C_VEL
LIN {X 0,Y 361.82,Z 84.913,A -85,B 0,C 180,E1 -13095.946,E2 -13095.946} C_VEL
LIN {X 0,Y 361.837,Z 84.904,A -85,B 0,C 180,E1 -13099.244,E2 -13099.244} C_VEL
LIN {X 0,Y 361.865,Z 84.91,A -85,B 0,C 180,E1 -13102.777,E2 -13102.777} C_VEL
LIN {X 0,Y 361.855,Z 84.892,A -85,B 0,C 180,E1 -13105.719,E2 -13105.719} C_VEL
LIN {X 0,Y 361.874,Z 84.906,A -85,B 0,C 180,E1 -13109.671,E2 -13109.671} C_VEL
LIN {X 0,Y 361.955,Z 84.878,A -85,B 0,C 180,E1 -13113.475,E2 -13113.475} C_VEL
LIN {X 0,Y 361.893,Z 84.904,A -85,B 0,C 180,E1 -13117.144,E2 -13117.144} C_VEL
LIN {X 0,Y 361.908,Z 84.877,A -85,B 0,C 180,E1 -13120.723,E2 -13120.723} C_VEL
LIN {X 0,Y 361.934,Z 84.889,A -85,B 0,C 180,E1 -13123.065,E2 -13123.065} C_VEL
LIN {X 0,Y 361.999,Z 84.889,A -85,B 0,C 180,E1 -13126.527,E2 -13126.527} C_VEL
LIN {X 0,Y 362.031,Z 84.86,A -85,B 0,C 180,E1 -13129.937,E2 -13129.937} C_VEL
LIN {X 0,Y 362.151,Z 84.857,A -85,B 0,C 180,E1 -13132.192,E2 -13132.192} C_VEL
LIN {X 0,Y 362.121,Z 84.879,A -85,B 0,C 180,E1 -13134.431,E2 -13134.431} C_VEL
LIN {X 0,Y 362.28,Z 84.846,A -85,B 0,C 180,E1 -13137.776,E2 -13137.776} C_VEL
LIN {X 0,Y 362.426,Z 84.81,A -85,B 0,C 180,E1 -13139.999,E2 -13139.999} C_VEL
LIN {X 0,Y 362.28,Z 84.845,A -85,B 0,C 180,E1 -13142.223,E2 -13142.223} C_VEL
LIN {X 0,Y 362.172,Z 84.865,A -85,B 0,C 180,E1 -13146.686,E2 -13146.686} C_VEL
LIN {X 0,Y 362.074,Z 84.86,A -85,B 0,C 180,E1 -13148.933,E2 -13148.933} C_VEL
LIN {X 0,Y 361.966,Z 84.89,A -85,B 0,C 180,E1 -13152.331,E2 -13152.331} C_VEL
LIN {X 0,Y 361.961,Z 84.896,A -85,B 0,C 180,E1 -13154.62,E2 -13154.62} C_VEL
LIN {X 0,Y 361.954,Z 84.876,A -85,B 0,C 180,E1 -13158.099,E2 -13158.099} C_VEL
LIN {X 0,Y 361.891,Z 84.903,A -85,B 0,C 180,E1 -13161.652,E2 -13161.652} C_VEL
LIN {X 0,Y 361.926,Z 84.893,A -85,B 0,C 180,E1 -13165.289,E2 -13165.289} C_VEL
LIN {X 0,Y 361.906,Z 84.886,A -85,B 0,C 180,E1 -13167.778,E2 -13167.778} C_VEL
LIN {X 0,Y 361.835,Z 84.912,A -85,B 0,C 180,E1 -13171.629,E2 -13171.629} C_VEL
LIN {X 0,Y 361.872,Z 84.898,A -85,B 0,C 180,E1 -13175.344,E2 -13175.344} C_VEL
LIN {X 0,Y 361.871,Z 84.904,A -85,B 0,C 180,E1 -13179.027,E2 -13179.027} C_VEL
LIN {X 0,Y 361.853,Z 84.908,A -85,B 0,C 180,E1 -13182.435,E2 -13182.435} C_VEL
LIN {X 0,Y 361.814,Z 84.894,A -85,B 0,C 180,E1 -13185.946,E2 -13185.946} C_VEL
LIN {X 0,Y 361.831,Z 84.883,A -85,B 0,C 180,E1 -13189.244,E2 -13189.244} C_VEL
LIN {X 0,Y 361.861,Z 84.907,A -85,B 0,C 180,E1 -13192.776,E2 -13192.776} C_VEL
LIN {X 0,Y 361.851,Z 84.884,A -85,B 0,C 180,E1 -13195.719,E2 -13195.719} C_VEL
LIN {X 0,Y 361.869,Z 84.897,A -85,B 0,C 180,E1 -13199.672,E2 -13199.672} C_VEL
LIN {X 0,Y 361.95,Z 84.901,A -85,B 0,C 180,E1 -13203.475,E2 -13203.475} C_VEL
LIN {X 0,Y 361.887,Z 84.909,A -85,B 0,C 180,E1 -13207.145,E2 -13207.145} C_VEL
LIN {X 0,Y 361.917,Z 84.905,A -85,B 0,C 180,E1 -13210.724,E2 -13210.724} C_VEL
LIN {X 0,Y 361.991,Z 85.166,A -85,B 0,C 180,E1 -13212.266,E2 -13212.266} C_VEL
LIN {X 0,Y 362.282,Z 86.408,A -85,B 0,C 180,E1 -13212.581,E2 -13212.581} C_VEL
LIN {X 0,Y 363.944,Z 89.048,A -85,B 0,C 180,E1 -13213.096,E2 -13213.096} C_VEL
LIN {X 0,Y 366.435,Z 90.945,A -85,B 0,C 180,E1 -13213.835,E2 -13213.835} C_VEL
LIN {X 0,Y 368.238,Z 93.827,A -85,B 0,C 180,E1 -13214.425,E2 -13214.425} C_VEL
LIN {X 0,Y 370.693,Z 95.955,A -85,B 0,C 180,E1 -13215.218,E2 -13215.218} C_VEL
LIN {X 0,Y 371.854,Z 96.828,A -85,B 0,C 180,E1 -13215.602,E2 -13215.602} C_VEL
LIN {X 0,Y 374.176,Z 100.035,A -85,B 0,C 180,E1 -13216.445,E2 -13216.445} C_VEL
LIN {X 0,Y 376.963,Z 102.256,A -85,B 0,C 180,E1 -13217.483,E2 -13217.483} C_VEL
LIN {X 0,Y 377.928,Z 103.055,A -85,B 0,C 180,E1 -13217.856,E2 -13217.856} C_VEL
LIN {X 0,Y 380.531,Z 106.38,A -85,B 0,C 180,E1 -13219.02,E2 -13219.02} C_VEL
LIN {X 0,Y 383.373,Z 108.501,A -85,B 0,C 180,E1 -13220.37,E2 -13220.37} C_VEL
LIN {X 0,Y 384.988,Z 109.445,A -85,B 0,C 180,E1 -13221.206,E2 -13221.206} C_VEL
LIN {X 0,Y 387.164,Z 112.426,A -85,B 0,C 180,E1 -13222.596,E2 -13222.596} C_VEL
LIN {X 0,Y 389.259,Z 114.251,A -85,B 0,C 180,E1 -13224.171,E2 -13224.171} C_VEL
LIN {X 0,Y 391.009,Z 115.289,A -85,B 0,C 180,E1 -13225.877,E2 -13225.877} C_VEL
LIN {X 0,Y 392.128,Z 115.663,A -85,B 0,C 180,E1 -13227.451,E2 -13227.451} C_VEL
LIN {X 0,Y 392.722,Z 116.119,A -85,B 0,C 180,E1 -13228.975,E2 -13228.975} C_VEL
LIN {X 0,Y 392.864,Z 116.021,A -85,B 0,C 180,E1 -13230,E2 -13230} C_VEL
LIN {X 0,Y 392.599,Z 115.97,A -85,B 0,C 180,E1 -13231.539,E2 -13231.539} C_VEL
LIN {X 0,Y 391.864,Z 115.542,A -85,B 0,C 180,E1 -13233.084,E2 -13233.084} C_VEL
LIN {X 0,Y 390.285,Z 114.928,A -85,B 0,C 180,E1 -13234.907,E2 -13234.907} C_VEL
LIN {X 0,Y 388.214,Z 113.473,A -85,B 0,C 180,E1 -13236.635,E2 -13236.635} C_VEL
LIN {X 0,Y 386.329,Z 111.397,A -85,B 0,C 180,E1 -13237.961,E2 -13237.961} C_VEL
LIN {X 0,Y 384.776,Z 109.127,A -85,B 0,C 180,E1 -13238.931,E2 -13238.931} C_VEL
LIN {X 0,Y 381.795,Z 107.488,A -85,B 0,C 180,E1 -13240.39,E2 -13240.39} C_VEL
LIN {X 0,Y 379.033,Z 104.745,A -85,B 0,C 180,E1 -13241.628,E2 -13241.628} C_VEL
LIN {X 0,Y 377.387,Z 102.464,A -85,B 0,C 180,E1 -13242.366,E2 -13242.366} C_VEL
LIN {X 0,Y 374.54,Z 100.421,A -85,B 0,C 180,E1 -13243.413,E2 -13243.413} C_VEL
LIN {X 0,Y 372.281,Z 97.503,A -85,B 0,C 180,E1 -13244.245,E2 -13244.245} C_VEL
LIN {X 0,Y 371.417,Z 96.364,A -85,B 0,C 180,E1 -13244.548,E2 -13244.548} C_VEL
LIN {X 0,Y 368.646,Z 94.258,A -85,B 0,C 180,E1 -13245.453,E2 -13245.453} C_VEL
LIN {X 0,Y 366.669,Z 91.428,A -85,B 0,C 180,E1 -13246.083,E2 -13246.083} C_VEL
LIN {X 0,Y 366.072,Z 90.534,A -85,B 0,C 180,E1 -13246.279,E2 -13246.279} C_VEL
LIN {X 0,Y 363.705,Z 88.798,A -85,B 0,C 180,E1 -13246.969,E2 -13246.969} C_VEL
LIN {X 0,Y 362.154,Z 85.984,A -85,B 0,C 180,E1 -13247.49,E2 -13247.49} C_VEL
LIN {X 0,Y 361.959,Z 85.006,A -85,B 0,C 180,E1 -13247.859,E2 -13247.859} C_VEL
LIN {X 0,Y 361.888,Z 84.909,A -85,B 0,C 180,E1 -13251.653,E2 -13251.653} C_VEL
LIN {X 0,Y 361.925,Z 84.903,A -85,B 0,C 180,E1 -13255.29,E2 -13255.29} C_VEL
LIN {X 0,Y 361.905,Z 84.9,A -85,B 0,C 180,E1 -13257.779,E2 -13257.779} C_VEL
LIN {X 0,Y 361.834,Z 84.914,A -85,B 0,C 180,E1 -13261.63,E2 -13261.63} C_VEL
LIN {X 0,Y 361.871,Z 84.881,A -85,B 0,C 180,E1 -13265.345,E2 -13265.345} C_VEL
LIN {X 0,Y 361.868,Z 84.908,A -85,B 0,C 180,E1 -13269.027,E2 -13269.027} C_VEL
LIN {X 0,Y 361.832,Z 84.875,A -85,B 0,C 180,E1 -13272.829,E2 -13272.829} C_VEL
LIN {X 0,Y 361.823,Z 84.915,A -85,B 0,C 180,E1 -13275.946,E2 -13275.946} C_VEL
LIN {X 0,Y 361.862,Z 84.898,A -85,B 0,C 180,E1 -13279.595,E2 -13279.595} C_VEL
LIN {X 0,Y 361.203,Z 84.985,A -85,B 0,C 180,E1 -13280.524,E2 -13280.524} C_VEL
LIN {X 0,Y 358.361,Z 85.346,A -85,B 0,C 180,E1 -13282.034,E2 -13282.034} C_VEL
LIN {X 0,Y 355.945,Z 85.646,A -85,B 0,C 180,E1 -13283.256,E2 -13283.256} C_VEL
LIN {X 0,Y 354.9,Z 85.77,A -85,B 0,C 180,E1 -13284.201,E2 -13284.201} C_VEL
LIN {X 0,Y 354.811,Z 85.778,A -85,B 0,C 180,E1 -13284.521,E2 -13284.521} C_VEL
LIN {X 0,Y 354.784,Z 85.791,A -85,B 0,C 180,E1 -13287.667,E2 -13287.667} C_VEL
LIN {X 0,Y 354.844,Z 85.768,A -85,B 0,C 180,E1 -13291.619,E2 -13291.619} C_VEL
LIN {X 0,Y 354.897,Z 85.764,A -85,B 0,C 180,E1 -13294.173,E2 -13294.173} C_VEL
LIN {X 0,Y 354.834,Z 85.782,A -85,B 0,C 180,E1 -13297.895,E2 -13297.895} C_VEL
LIN {X 0,Y 354.921,Z 85.752,A -85,B 0,C 180,E1 -13301.892,E2 -13301.892} C_VEL
LIN {X 0,Y 354.942,Z 85.771,A -85,B 0,C 180,E1 -13305.981,E2 -13305.981} C_VEL
LIN {X 0,Y 354.98,Z 85.739,A -85,B 0,C 180,E1 -13309.737,E2 -13309.737} C_VEL
LIN {X 0,Y 355.113,Z 85.733,A -85,B 0,C 180,E1 -13312.037,E2 -13312.037} C_VEL
LIN {X 0,Y 355.092,Z 85.754,A -85,B 0,C 180,E1 -13314.321,E2 -13314.321} C_VEL
LIN {X 0,Y 355.243,Z 85.721,A -85,B 0,C 180,E1 -13317.733,E2 -13317.733} C_VEL
LIN {X 0,Y 355.375,Z 85.687,A -85,B 0,C 180,E1 -13320.001,E2 -13320.001} C_VEL
LIN {X 0,Y 355.243,Z 85.723,A -85,B 0,C 180,E1 -13322.268,E2 -13322.268} C_VEL
LIN {X 0,Y 355.142,Z 85.739,A -85,B 0,C 180,E1 -13326.82,E2 -13326.82} C_VEL
LIN {X 0,Y 355.016,Z 85.735,A -85,B 0,C 180,E1 -13329.113,E2 -13329.113} C_VEL
LIN {X 0,Y 354.922,Z 85.766,A -85,B 0,C 180,E1 -13332.581,E2 -13332.581} C_VEL
LIN {X 0,Y 354.89,Z 85.768,A -85,B 0,C 180,E1 -13336.097,E2 -13336.097} C_VEL
LIN {X 0,Y 354.902,Z 85.748,A -85,B 0,C 180,E1 -13338.473,E2 -13338.473} C_VEL
LIN {X 0,Y 354.837,Z 85.781,A -85,B 0,C 180,E1 -13342.106,E2 -13342.106} C_VEL
LIN {X 0,Y 354.9,Z 85.76,A -85,B 0,C 180,E1 -13345.828,E2 -13345.828} C_VEL
LIN {X 0,Y 354.819,Z 85.785,A -85,B 0,C 180,E1 -13349.682,E2 -13349.682} C_VEL
LIN {X 0,Y 354.807,Z 85.771,A -85,B 0,C 180,E1 -13353.703,E2 -13353.703} C_VEL
LIN {X 0,Y 354.799,Z 85.786,A -85,B 0,C 180,E1 -13356.46,E2 -13356.46} C_VEL
LIN {X 0,Y 354.826,Z 85.775,A -85,B 0,C 180,E1 -13359.424,E2 -13359.424} C_VEL
LIN {X 0,Y 354.79,Z 85.792,A -85,B 0,C 180,E1 -13362.868,E2 -13362.868} C_VEL
LIN {X 0,Y 354.769,Z 85.791,A -85,B 0,C 180,E1 -13366.104,E2 -13366.104} C_VEL
LIN {X 0,Y 354.789,Z 85.769,A -85,B 0,C 180,E1 -13369.179,E2 -13369.179} C_VEL
LIN {X 0,Y 354.814,Z 85.79,A -85,B 0,C 180,E1 -13372.402,E2 -13372.402} C_VEL
LIN {X 0,Y 354.814,Z 85.773,A -85,B 0,C 180,E1 -13374.941,E2 -13374.941} C_VEL
LIN {X 0,Y 354.883,Z 85.887,A -85,B 0,C 180,E1 -13378.081,E2 -13378.081} C_VEL
LIN {X 0,Y 356.407,Z 93.486,A -85,B 0,C 180,E1 -13380.788,E2 -13380.788} C_VEL
LIN {X 0,Y 357.867,Z 101.849,A -85,B 0,C 180,E1 -13383.463,E2 -13383.463} C_VEL
LIN {X 0,Y 357.815,Z 105.589,A -85,B 0,C 180,E1 -13384.624,E2 -13384.624} C_VEL
LIN {X 0,Y 356.758,Z 114.709,A -85,B 0,C 180,E1 -13387.388,E2 -13387.388} C_VEL
LIN {X 0,Y 357.92,Z 120.343,A -85,B 0,C 180,E1 -13387.638,E2 -13387.638} C_VEL
LIN {X 0,Y 362.841,Z 145.942,A -85,B 0,C 180,E1 -13388.488,E2 -13388.488} C_VEL
LIN {X 0,Y 363.451,Z 152.131,A -85,B 0,C 180,E1 -13388.654,E2 -13388.654} C_VEL
LIN {X 0,Y 362.334,Z 219.494,A -85,B 0,C 180,E1 -13390.01,E2 -13390.01} C_VEL
LIN {X 0,Y 361.851,Z 230.25,A -85,B 0,C 180,E1 -13390.352,E2 -13390.352} C_VEL
LIN {X 0,Y 361.235,Z 239.35,A -85,B 0,C 180,E1 -13390.76,E2 -13390.76} C_VEL
LIN {X 0,Y 360.472,Z 249.712,A -85,B 0,C 180,E1 -13391.382,E2 -13391.382} C_VEL
LIN {X 0,Y 359.617,Z 258.844,A -85,B 0,C 180,E1 -13392.073,E2 -13392.073} C_VEL
LIN {X 0,Y 358.722,Z 267.84,A -85,B 0,C 180,E1 -13392.91,E2 -13392.91} C_VEL
LIN {X 0,Y 357.749,Z 276.567,A -85,B 0,C 180,E1 -13393.89,E2 -13393.89} C_VEL
LIN {X 0,Y 356.916,Z 284.392,A -85,B 0,C 180,E1 -13394.942,E2 -13394.942} C_VEL
LIN {X 0,Y 355.988,Z 292.81,A -85,B 0,C 180,E1 -13396.296,E2 -13396.296} C_VEL
LIN {X 0,Y 355.303,Z 298.761,A -85,B 0,C 180,E1 -13397.433,E2 -13397.433} C_VEL
LIN {X 0,Y 354.522,Z 305.076,A -85,B 0,C 180,E1 -13398.856,E2 -13398.856} C_VEL
LIN {X 0,Y 354.025,Z 310.339,A -85,B 0,C 180,E1 -13400.286,E2 -13400.286} C_VEL
LIN {X 0,Y 353.612,Z 315.47,A -85,B 0,C 180,E1 -13402.003,E2 -13402.003} C_VEL
LIN {X 0,Y 353.417,Z 318.241,A -85,B 0,C 180,E1 -13403.147,E2 -13403.147} C_VEL
LIN {X 0,Y 353.291,Z 320.608,A -85,B 0,C 180,E1 -13404.292,E2 -13404.292} C_VEL
LIN {X 0,Y 353.263,Z 322.408,A -85,B 0,C 180,E1 -13405.436,E2 -13405.436} C_VEL
LIN {X 0,Y 353.172,Z 324.852,A -85,B 0,C 180,E1 -13407.719,E2 -13407.719} C_VEL
LIN {X 0,Y 353.204,Z 325.442,A -85,B 0,C 180,E1 -13408.86,E2 -13408.86} C_VEL
LIN {X 0,Y 353.263,Z 325.598,A -85,B 0,C 180,E1 -13410,E2 -13410} C_VEL
LIN {X 0,Y 353.204,Z 325.442,A -85,B 0,C 180,E1 -13411.14,E2 -13411.14} C_VEL
LIN {X 0,Y 353.172,Z 324.852,A -85,B 0,C 180,E1 -13412.281,E2 -13412.281} C_VEL
LIN {X 0,Y 353.261,Z 322.408,A -85,B 0,C 180,E1 -13414.564,E2 -13414.564} C_VEL
LIN {X 0,Y 353.336,Z 319.459,A -85,B 0,C 180,E1 -13416.28,E2 -13416.28} C_VEL
LIN {X 0,Y 353.612,Z 315.47,A -85,B 0,C 180,E1 -13417.997,E2 -13417.997} C_VEL
LIN {X 0,Y 354.025,Z 310.339,A -85,B 0,C 180,E1 -13419.714,E2 -13419.714} C_VEL
LIN {X 0,Y 354.522,Z 305.076,A -85,B 0,C 180,E1 -13421.144,E2 -13421.144} C_VEL
LIN {X 0,Y 355.307,Z 298.762,A -85,B 0,C 180,E1 -13422.567,E2 -13422.567} C_VEL
LIN {X 0,Y 355.994,Z 292.811,A -85,B 0,C 180,E1 -13423.704,E2 -13423.704} C_VEL
LIN {X 0,Y 356.807,Z 285.884,A -85,B 0,C 180,E1 -13424.836,E2 -13424.836} C_VEL
LIN {X 0,Y 357.669,Z 277.703,A -85,B 0,C 180,E1 -13425.967,E2 -13425.967} C_VEL
LIN {X 0,Y 358.563,Z 269.191,A -85,B 0,C 180,E1 -13426.951,E2 -13426.951} C_VEL
LIN {X 0,Y 359.478,Z 260.477,A -85,B 0,C 180,E1 -13427.787,E2 -13427.787} C_VEL
LIN {X 0,Y 360.369,Z 250.719,A -85,B 0,C 180,E1 -13428.55,E2 -13428.55} C_VEL
LIN {X 0,Y 361.053,Z 241.925,A -85,B 0,C 180,E1 -13429.102,E2 -13429.102} C_VEL
LIN {X 0,Y 361.736,Z 231.998,A -85,B 0,C 180,E1 -13429.581,E2 -13429.581} C_VEL
LIN {X 0,Y 362.217,Z 222.143,A -85,B 0,C 180,E1 -13429.923,E2 -13429.923} C_VEL
LIN {X 0,Y 362.757,Z 197.021,A -85,B 0,C 180,E1 -13430.457,E2 -13430.457} C_VEL
LIN {X 0,Y 363.405,Z 149.705,A -85,B 0,C 180,E1 -13431.399,E2 -13431.399} C_VEL
LIN {X 0,Y 358.605,Z 123.524,A -85,B 0,C 180,E1 -13432.25,E2 -13432.25} C_VEL
LIN {X 0,Y 356.742,Z 114.908,A -85,B 0,C 180,E1 -13432.588,E2 -13432.588} C_VEL
LIN {X 0,Y 356.922,Z 112.643,A -85,B 0,C 180,E1 -13433.192,E2 -13433.192} C_VEL
LIN {X 0,Y 358.018,Z 102.909,A -85,B 0,C 180,E1 -13436.211,E2 -13436.211} C_VEL
LIN {X 0,Y 356.896,Z 95.849,A -85,B 0,C 180,E1 -13438.524,E2 -13438.524} C_VEL
LIN {X 0,Y 354.862,Z 85.819,A -85,B 0,C 180,E1 -13441.971,E2 -13441.971} C_VEL
LIN {X 0,Y 354.825,Z 85.773,A -85,B 0,C 180,E1 -13445.699,E2 -13445.699} C_VEL
LIN {X 0,Y 354.826,Z 85.765,A -85,B 0,C 180,E1 -13449.423,E2 -13449.423} C_VEL
LIN {X 0,Y 354.79,Z 85.79,A -85,B 0,C 180,E1 -13452.867,E2 -13452.867} C_VEL
LIN {X 0,Y 354.769,Z 85.792,A -85,B 0,C 180,E1 -13456.103,E2 -13456.103} C_VEL
LIN {X 0,Y 354.789,Z 85.782,A -85,B 0,C 180,E1 -13459.178,E2 -13459.178} C_VEL
LIN {X 0,Y 354.808,Z 85.787,A -85,B 0,C 180,E1 -13462.402,E2 -13462.402} C_VEL
LIN {X 0,Y 354.813,Z 85.774,A -85,B 0,C 180,E1 -13464.94,E2 -13464.94} C_VEL
LIN {X 0,Y 354.794,Z 85.787,A -85,B 0,C 180,E1 -13468.405,E2 -13468.405} C_VEL
LIN {X 0,Y 354.847,Z 85.77,A -85,B 0,C 180,E1 -13471.618,E2 -13471.618} C_VEL
LIN {X 0,Y 354.9,Z 85.76,A -85,B 0,C 180,E1 -13474.172,E2 -13474.172} C_VEL
LIN {X 0,Y 354.837,Z 85.781,A -85,B 0,C 180,E1 -13477.894,E2 -13477.894} C_VEL
LIN {X 0,Y 354.923,Z 85.747,A -85,B 0,C 180,E1 -13481.891,E2 -13481.891} C_VEL
LIN {X 0,Y 354.943,Z 85.769,A -85,B 0,C 180,E1 -13485.981,E2 -13485.981} C_VEL
LIN {X 0,Y 354.978,Z 85.739,A -85,B 0,C 180,E1 -13489.735,E2 -13489.735} C_VEL
LIN {X 0,Y 355.114,Z 85.731,A -85,B 0,C 180,E1 -13492.036,E2 -13492.036} C_VEL
LIN {X 0,Y 355.096,Z 85.754,A -85,B 0,C 180,E1 -13494.32,E2 -13494.32} C_VEL
LIN {X 0,Y 355.243,Z 85.723,A -85,B 0,C 180,E1 -13497.732,E2 -13497.732} C_VEL
LIN {X 0,Y 355.375,Z 85.687,A -85,B 0,C 180,E1 -13499.999,E2 -13499.999} C_VEL
LIN {X 0,Y 355.243,Z 85.721,A -85,B 0,C 180,E1 -13502.267,E2 -13502.267} C_VEL
LIN {X 0,Y 355.138,Z 85.741,A -85,B 0,C 180,E1 -13506.819,E2 -13506.819} C_VEL
LIN {X 0,Y 355.015,Z 85.736,A -85,B 0,C 180,E1 -13509.112,E2 -13509.112} C_VEL
LIN {X 0,Y 354.925,Z 85.766,A -85,B 0,C 180,E1 -13512.58,E2 -13512.58} C_VEL
LIN {X 0,Y 354.889,Z 85.772,A -85,B 0,C 180,E1 -13516.095,E2 -13516.095} C_VEL
LIN {X 0,Y 354.9,Z 85.753,A -85,B 0,C 180,E1 -13518.471,E2 -13518.471} C_VEL
LIN {X 0,Y 354.834,Z 85.782,A -85,B 0,C 180,E1 -13522.105,E2 -13522.105} C_VEL
LIN {X 0,Y 354.897,Z 85.764,A -85,B 0,C 180,E1 -13525.827,E2 -13525.827} C_VEL
LIN {X 0,Y 354.815,Z 85.785,A -85,B 0,C 180,E1 -13529.681,E2 -13529.681} C_VEL
LIN {X 0,Y 354.803,Z 85.775,A -85,B 0,C 180,E1 -13533.701,E2 -13533.701} C_VEL
LIN {X 0,Y 354.796,Z 85.786,A -85,B 0,C 180,E1 -13536.459,E2 -13536.459} C_VEL
LIN {X 0,Y 354.821,Z 85.78,A -85,B 0,C 180,E1 -13539.423,E2 -13539.423} C_VEL
LIN {X 0,Y 354.801,Z 85.791,A -85,B 0,C 180,E1 -13542.87,E2 -13542.87} C_VEL
LIN {X 0,Y 354.763,Z 85.768,A -85,B 0,C 180,E1 -13546.103,E2 -13546.103} C_VEL
LIN {X 0,Y 354.783,Z 85.759,A -85,B 0,C 180,E1 -13549.179,E2 -13549.179} C_VEL
LIN {X 0,Y 354.805,Z 85.79,A -85,B 0,C 180,E1 -13552.402,E2 -13552.402} C_VEL
LIN {X 0,Y 354.808,Z 85.76,A -85,B 0,C 180,E1 -13554.941,E2 -13554.941} C_VEL
LIN {X 0,Y 354.79,Z 85.792,A -85,B 0,C 180,E1 -13558.405,E2 -13558.405} C_VEL
LIN {X 0,Y 354.843,Z 85.77,A -85,B 0,C 180,E1 -13561.618,E2 -13561.618} C_VEL
LIN {X 0,Y 354.895,Z 85.78,A -85,B 0,C 180,E1 -13564.172,E2 -13564.172} C_VEL
LIN {X 0,Y 354.831,Z 85.788,A -85,B 0,C 180,E1 -13567.894,E2 -13567.894} C_VEL
LIN {X 0,Y 354.913,Z 86.03,A -85,B 0,C 180,E1 -13570.667,E2 -13570.667} C_VEL
LIN {X 0,Y 355.228,Z 87.265,A -85,B 0,C 180,E1 -13570.969,E2 -13570.969} C_VEL
LIN {X 0,Y 356.951,Z 89.98,A -85,B 0,C 180,E1 -13571.466,E2 -13571.466} C_VEL
LIN {X 0,Y 359.108,Z 91.684,A -85,B 0,C 180,E1 -13572.017,E2 -13572.017} C_VEL
LIN {X 0,Y 361.197,Z 94.981,A -85,B 0,C 180,E1 -13572.647,E2 -13572.647} C_VEL
LIN {X 0,Y 364.119,Z 97.435,A -85,B 0,C 180,E1 -13573.452,E2 -13573.452} C_VEL
LIN {X 0,Y 366.534,Z 100.723,A -85,B 0,C 180,E1 -13574.233,E2 -13574.233} C_VEL
LIN {X 0,Y 369.929,Z 103.533,A -85,B 0,C 180,E1 -13575.301,E2 -13575.301} C_VEL
LIN {X 0,Y 372.825,Z 107.08,A -85,B 0,C 180,E1 -13576.312,E2 -13576.312} C_VEL
LIN {X 0,Y 376.19,Z 109.732,A -85,B 0,C 180,E1 -13577.559,E2 -13577.559} C_VEL
LIN {X 0,Y 379.015,Z 113.135,A -85,B 0,C 180,E1 -13578.786,E2 -13578.786} C_VEL
LIN {X 0,Y 381.764,Z 115.214,A -85,B 0,C 180,E1 -13580.044,E2 -13580.044} C_VEL
LIN {X 0,Y 383.693,Z 116.296,A -85,B 0,C 180,E1 -13580.976,E2 -13580.976} C_VEL
LIN {X 0,Y 386.24,Z 119.578,A -85,B 0,C 180,E1 -13582.578,E2 -13582.578} C_VEL
LIN {X 0,Y 388.479,Z 121.425,A -85,B 0,C 180,E1 -13584.266,E2 -13584.266} C_VEL
LIN {X 0,Y 390.135,Z 122.329,A -85,B 0,C 180,E1 -13585.868,E2 -13585.868} C_VEL
LIN {X 0,Y 391.261,Z 122.71,A -85,B 0,C 180,E1 -13587.445,E2 -13587.445} C_VEL
LIN {X 0,Y 391.857,Z 123.165,A -85,B 0,C 180,E1 -13588.972,E2 -13588.972} C_VEL
LIN {X 0,Y 391.999,Z 123.068,A -85,B 0,C 180,E1 -13590,E2 -13590} C_VEL
LIN {X 0,Y 391.73,Z 123.017,A -85,B 0,C 180,E1 -13591.542,E2 -13591.542} C_VEL
LIN {X 0,Y 390.988,Z 122.588,A -85,B 0,C 180,E1 -13593.091,E2 -13593.091} C_VEL
LIN {X 0,Y 389.394,Z 121.972,A -85,B 0,C 180,E1 -13594.918,E2 -13594.918} C_VEL
LIN {X 0,Y 387.3,Z 120.54,A -85,B 0,C 180,E1 -13596.652,E2 -13596.652} C_VEL
LIN {X 0,Y 385.253,Z 118.467,A -85,B 0,C 180,E1 -13598.052,E2 -13598.052} C_VEL
LIN {X 0,Y 383.438,Z 116.004,A -85,B 0,C 180,E1 -13599.167,E2 -13599.167} C_VEL
LIN {X 0,Y 380.179,Z 114.107,A -85,B 0,C 180,E1 -13600.72,E2 -13600.72} C_VEL
LIN {X 0,Y 377.084,Z 110.938,A -85,B 0,C 180,E1 -13602.069,E2 -13602.069} C_VEL
LIN {X 0,Y 375.687,Z 109.209,A -85,B 0,C 180,E1 -13602.629,E2 -13602.629} C_VEL
LIN {X 0,Y 372.662,Z 106.885,A -85,B 0,C 180,E1 -13603.749,E2 -13603.749} C_VEL
LIN {X 0,Y 369.992,Z 103.66,A -85,B 0,C 180,E1 -13604.675,E2 -13604.675} C_VEL
LIN {X 0,Y 368.942,Z 102.624,A -85,B 0,C 180,E1 -13605.039,E2 -13605.039} C_VEL
LIN {X 0,Y 365.921,Z 100.078,A -85,B 0,C 180,E1 -13605.956,E2 -13605.956} C_VEL
LIN {X 0,Y 363.644,Z 96.894,A -85,B 0,C 180,E1 -13606.693,E2 -13606.693} C_VEL
LIN {X 0,Y 360.934,Z 94.666,A -85,B 0,C 180,E1 -13607.427,E2 -13607.427} C_VEL
LIN {X 0,Y 358.716,Z 91.214,A -85,B 0,C 180,E1 -13608.097,E2 -13608.097} C_VEL
LIN {X 0,Y 356.498,Z 89.471,A -85,B 0,C 180,E1 -13608.649,E2 -13608.649} C_VEL
LIN {X 0,Y 355.028,Z 86.603,A -85,B 0,C 180,E1 -13609.14,E2 -13609.14} C_VEL
LIN {X 0,Y 354.861,Z 85.836,A -85,B 0,C 180,E1 -13609.524,E2 -13609.524} C_VEL
LIN {X 0,Y 354.829,Z 85.788,A -85,B 0,C 180,E1 -13613.337,E2 -13613.337} C_VEL
LIN {X 0,Y 354.884,Z 85.78,A -85,B 0,C 180,E1 -13616.982,E2 -13616.982} C_VEL
LIN {X 0,Y 354.814,Z 85.769,A -85,B 0,C 180,E1 -13619.682,E2 -13619.682} C_VEL
LIN {X 0,Y 354.81,Z 85.763,A -85,B 0,C 180,E1 -13623.684,E2 -13623.684} C_VEL
LIN {X 0,Y 354.796,Z 85.78,A -85,B 0,C 180,E1 -13626.46,E2 -13626.46} C_VEL
LIN {X 0,Y 354.82,Z 85.778,A -85,B 0,C 180,E1 -13629.424,E2 -13629.424} C_VEL
LIN {X 0,Y 354.784,Z 85.752,A -85,B 0,C 180,E1 -13632.867,E2 -13632.867} C_VEL
LIN {X 0,Y 354.772,Z 85.793,A -85,B 0,C 180,E1 -13636.105,E2 -13636.105} C_VEL
LIN {X 0,Y 354.799,Z 85.776,A -85,B 0,C 180,E1 -13639.589,E2 -13639.589} C_VEL
LIN {X 0,Y 354.806,Z 85.788,A -85,B 0,C 180,E1 -13642.403,E2 -13642.403} C_VEL
LIN {X 0,Y 354.811,Z 85.778,A -85,B 0,C 180,E1 -13644.521,E2 -13644.521} C_VEL
LIN {X 0,Y 354.121,Z 85.859,A -85,B 0,C 180,E1 -13645.468,E2 -13645.468} C_VEL
LIN {X 0,Y 351.225,Z 86.225,A -85,B 0,C 180,E1 -13647.007,E2 -13647.007} C_VEL
LIN {X 0,Y 348.805,Z 86.534,A -85,B 0,C 180,E1 -13648.253,E2 -13648.253} C_VEL
LIN {X 0,Y 347.802,Z 86.663,A -85,B 0,C 180,E1 -13649.218,E2 -13649.218} C_VEL
LIN {X 0,Y 347.739,Z 86.666,A -85,B 0,C 180,E1 -13649.545,E2 -13649.545} C_VEL
LIN {X 0,Y 347.848,Z 86.634,A -85,B 0,C 180,E1 -13652.746,E2 -13652.746} C_VEL
LIN {X 0,Y 347.787,Z 86.661,A -85,B 0,C 180,E1 -13656.163,E2 -13656.163} C_VEL
LIN {X 0,Y 347.811,Z 86.641,A -85,B 0,C 180,E1 -13659.91,E2 -13659.91} C_VEL
LIN {X 0,Y 347.865,Z 86.633,A -85,B 0,C 180,E1 -13662.36,E2 -13662.36} C_VEL
LIN {X 0,Y 347.896,Z 86.649,A -85,B 0,C 180,E1 -13665.971,E2 -13665.971} C_VEL
LIN {X 0,Y 347.931,Z 86.618,A -85,B 0,C 180,E1 -13669.526,E2 -13669.526} C_VEL
LIN {X 0,Y 348.074,Z 86.608,A -85,B 0,C 180,E1 -13671.875,E2 -13671.875} C_VEL
LIN {X 0,Y 348.067,Z 86.628,A -85,B 0,C 180,E1 -13674.206,E2 -13674.206} C_VEL
LIN {X 0,Y 348.206,Z 86.598,A -85,B 0,C 180,E1 -13677.687,E2 -13677.687} C_VEL
LIN {X 0,Y 348.325,Z 86.564,A -85,B 0,C 180,E1 -13680.001,E2 -13680.001} C_VEL
LIN {X 0,Y 348.206,Z 86.599,A -85,B 0,C 180,E1 -13682.314,E2 -13682.314} C_VEL
LIN {X 0,Y 348.109,Z 86.615,A -85,B 0,C 180,E1 -13686.958,E2 -13686.958} C_VEL
LIN {X 0,Y 347.968,Z 86.61,A -85,B 0,C 180,E1 -13689.299,E2 -13689.299} C_VEL
LIN {X 0,Y 347.891,Z 86.642,A -85,B 0,C 180,E1 -13692.84,E2 -13692.84} C_VEL
LIN {X 0,Y 347.84,Z 86.645,A -85,B 0,C 180,E1 -13696.432,E2 -13696.432} C_VEL
LIN {X 0,Y 347.852,Z 86.625,A -85,B 0,C 180,E1 -13698.861,E2 -13698.861} C_VEL
LIN {X 0,Y 347.776,Z 86.66,A -85,B 0,C 180,E1 -13702.58,E2 -13702.58} C_VEL
LIN {X 0,Y 347.813,Z 86.649,A -85,B 0,C 180,E1 -13705.109,E2 -13705.109} C_VEL
LIN {X 0,Y 347.809,Z 86.641,A -85,B 0,C 180,E1 -13707.695,E2 -13707.695} C_VEL
LIN {X 0,Y 347.75,Z 86.666,A -85,B 0,C 180,E1 -13710.348,E2 -13710.348} C_VEL
LIN {X 0,Y 347.749,Z 86.648,A -85,B 0,C 180,E1 -13714.044,E2 -13714.044} C_VEL
LIN {X 0,Y 347.763,Z 86.666,A -85,B 0,C 180,E1 -13717.321,E2 -13717.321} C_VEL
LIN {X 0,Y 347.733,Z 86.657,A -85,B 0,C 180,E1 -13720.298,E2 -13720.298} C_VEL
LIN {X 0,Y 347.725,Z 86.669,A -85,B 0,C 180,E1 -13723.409,E2 -13723.409} C_VEL
LIN {X 0,Y 347.727,Z 86.673,A -85,B 0,C 180,E1 -13726.687,E2 -13726.687} C_VEL
LIN {X 0,Y 347.749,Z 86.643,A -85,B 0,C 180,E1 -13730.174,E2 -13730.174} C_VEL
LIN {X 0,Y 347.768,Z 86.666,A -85,B 0,C 180,E1 -13732.68,E2 -13732.68} C_VEL
LIN {X 0,Y 347.751,Z 86.663,A -85,B 0,C 180,E1 -13735.957,E2 -13735.957} C_VEL
LIN {X 0,Y 347.801,Z 86.754,A -85,B 0,C 180,E1 -13737.702,E2 -13737.702} C_VEL
LIN {X 0,Y 349.421,Z 94.647,A -85,B 0,C 180,E1 -13740.571,E2 -13740.571} C_VEL
LIN {X 0,Y 350.859,Z 102.717,A -85,B 0,C 180,E1 -13743.212,E2 -13743.212} C_VEL
LIN {X 0,Y 350.906,Z 106.134,A -85,B 0,C 180,E1 -13744.326,E2 -13744.326} C_VEL
LIN {X 0,Y 349.892,Z 114.473,A -85,B 0,C 180,E1 -13746.911,E2 -13746.911} C_VEL
LIN {X 0,Y 350.721,Z 118.693,A -85,B 0,C 180,E1 -13747.122,E2 -13747.122} C_VEL
LIN {X 0,Y 355.372,Z 142.208,A -85,B 0,C 180,E1 -13747.938,E2 -13747.938} C_VEL
LIN {X 0,Y 356.861,Z 151.941,A -85,B 0,C 180,E1 -13748.24,E2 -13748.24} C_VEL
LIN {X 0,Y 355.676,Z 219.31,A -85,B 0,C 180,E1 -13749.619,E2 -13749.619} C_VEL
LIN {X 0,Y 355.186,Z 230.06,A -85,B 0,C 180,E1 -13749.967,E2 -13749.967} C_VEL
LIN {X 0,Y 354.554,Z 239.159,A -85,B 0,C 180,E1 -13750.383,E2 -13750.383} C_VEL
LIN {X 0,Y 353.721,Z 249.521,A -85,B 0,C 180,E1 -13751.013,E2 -13751.013} C_VEL
LIN {X 0,Y 352.875,Z 258.654,A -85,B 0,C 180,E1 -13751.719,E2 -13751.719} C_VEL
LIN {X 0,Y 351.922,Z 267.649,A -85,B 0,C 180,E1 -13752.569,E2 -13752.569} C_VEL
LIN {X 0,Y 350.899,Z 276.376,A -85,B 0,C 180,E1 -13753.567,E2 -13753.567} C_VEL
LIN {X 0,Y 350.065,Z 283.351,A -85,B 0,C 180,E1 -13754.508,E2 -13754.508} C_VEL
LIN {X 0,Y 349.233,Z 290.991,A -85,B 0,C 180,E1 -13755.728,E2 -13755.728} C_VEL
LIN {X 0,Y 348.52,Z 297.194,A -85,B 0,C 180,E1 -13756.888,E2 -13756.888} C_VEL
LIN {X 0,Y 347.671,Z 303.729,A -85,B 0,C 180,E1 -13758.338,E2 -13758.338} C_VEL
LIN {X 0,Y 347.235,Z 308.233,A -85,B 0,C 180,E1 -13759.504,E2 -13759.504} C_VEL
LIN {X 0,Y 346.681,Z 313.725,A -85,B 0,C 180,E1 -13761.255,E2 -13761.255} C_VEL
LIN {X 0,Y 346.344,Z 318.05,A -85,B 0,C 180,E1 -13763.007,E2 -13763.007} C_VEL
LIN {X 0,Y 346.203,Z 320.417,A -85,B 0,C 180,E1 -13764.174,E2 -13764.174} C_VEL
LIN {X 0,Y 346.161,Z 322.217,A -85,B 0,C 180,E1 -13765.342,E2 -13765.342} C_VEL
LIN {X 0,Y 346.084,Z 324.662,A -85,B 0,C 180,E1 -13767.672,E2 -13767.672} C_VEL
LIN {X 0,Y 346.104,Z 325.251,A -85,B 0,C 180,E1 -13768.836,E2 -13768.836} C_VEL
LIN {X 0,Y 346.165,Z 325.407,A -85,B 0,C 180,E1 -13770,E2 -13770} C_VEL
LIN {X 0,Y 346.104,Z 325.251,A -85,B 0,C 180,E1 -13771.164,E2 -13771.164} C_VEL
LIN {X 0,Y 346.084,Z 324.662,A -85,B 0,C 180,E1 -13772.328,E2 -13772.328} C_VEL
LIN {X 0,Y 346.159,Z 322.217,A -85,B 0,C 180,E1 -13774.658,E2 -13774.658} C_VEL
LIN {X 0,Y 346.263,Z 319.268,A -85,B 0,C 180,E1 -13776.409,E2 -13776.409} C_VEL
LIN {X 0,Y 346.552,Z 315.279,A -85,B 0,C 180,E1 -13778.161,E2 -13778.161} C_VEL
LIN {X 0,Y 347.008,Z 310.148,A -85,B 0,C 180,E1 -13779.913,E2 -13779.913} C_VEL
LIN {X 0,Y 347.522,Z 304.885,A -85,B 0,C 180,E1 -13781.372,E2 -13781.372} C_VEL
LIN {X 0,Y 348.351,Z 298.57,A -85,B 0,C 180,E1 -13782.822,E2 -13782.822} C_VEL
LIN {X 0,Y 349.058,Z 292.619,A -85,B 0,C 180,E1 -13783.982,E2 -13783.982} C_VEL
LIN {X 0,Y 350.061,Z 284.504,A -85,B 0,C 180,E1 -13785.314,E2 -13785.314} C_VEL
LIN {X 0,Y 350.943,Z 276.377,A -85,B 0,C 180,E1 -13786.431,E2 -13786.431} C_VEL
LIN {X 0,Y 351.912,Z 267.649,A -85,B 0,C 180,E1 -13787.431,E2 -13787.431} C_VEL
LIN {X 0,Y 352.888,Z 258.654,A -85,B 0,C 180,E1 -13788.281,E2 -13788.281} C_VEL
LIN {X 0,Y 353.822,Z 248.514,A -85,B 0,C 180,E1 -13789.056,E2 -13789.056} C_VEL
LIN {X 0,Y 354.677,Z 237.873,A -85,B 0,C 180,E1 -13789.686,E2 -13789.686} C_VEL
LIN {X 0,Y 355.485,Z 224.594,A -85,B 0,C 180,E1 -13790.241,E2 -13790.241} C_VEL
LIN {X 0,Y 356.015,Z 206.293,A -85,B 0,C 180,E1 -13790.663,E2 -13790.663} C_VEL
LIN {X 0,Y 356.821,Z 150.895,A -85,B 0,C 180,E1 -13791.784,E2 -13791.784} C_VEL
LIN {X 0,Y 352.178,Z 125.292,A -85,B 0,C 180,E1 -13792.636,E2 -13792.636} C_VEL
LIN {X 0,Y 349.888,Z 114.848,A -85,B 0,C 180,E1 -13793.044,E2 -13793.044} C_VEL
LIN {X 0,Y 349.918,Z 113.742,A -85,B 0,C 180,E1 -13793.261,E2 -13793.261} C_VEL
LIN {X 0,Y 351.013,Z 104.691,A -85,B 0,C 180,E1 -13796.135,E2 -13796.135} C_VEL
LIN {X 0,Y 350.294,Z 99.028,A -85,B 0,C 180,E1 -13798.02,E2 -13798.02} C_VEL
LIN {X 0,Y 348.185,Z 88.474,A -85,B 0,C 180,E1 -13801.655,E2 -13801.655} C_VEL
LIN {X 0,Y 347.801,Z 86.747,A -85,B 0,C 180,E1 -13802.298,E2 -13802.298} C_VEL
LIN {X 0,Y 347.774,Z 86.653,A -85,B 0,C 180,E1 -13806.065,E2 -13806.065} C_VEL
LIN {X 0,Y 347.755,Z 86.653,A -85,B 0,C 180,E1 -13808.792,E2 -13808.792} C_VEL
LIN {X 0,Y 347.753,Z 86.657,A -85,B 0,C 180,E1 -13811.83,E2 -13811.83} C_VEL
LIN {X 0,Y 347.707,Z 86.666,A -85,B 0,C 180,E1 -13815.026,E2 -13815.026} C_VEL
LIN {X 0,Y 347.752,Z 86.665,A -85,B 0,C 180,E1 -13818.397,E2 -13818.397} C_VEL
LIN {X 0,Y 347.774,Z 86.663,A -85,B 0,C 180,E1 -13822.011,E2 -13822.011} C_VEL
LIN {X 0,Y 347.746,Z 86.649,A -85,B 0,C 180,E1 -13825.536,E2 -13825.536} C_VEL
LIN {X 0,Y 347.746,Z 86.665,A -85,B 0,C 180,E1 -13828.3,E2 -13828.3} C_VEL
LIN {X 0,Y 347.78,Z 86.655,A -85,B 0,C 180,E1 -13830.987,E2 -13830.987} C_VEL
LIN {X 0,Y 347.832,Z 86.637,A -85,B 0,C 180,E1 -13833.607,E2 -13833.607} C_VEL
LIN {X 0,Y 347.79,Z 86.658,A -85,B 0,C 180,E1 -13836.161,E2 -13836.161} C_VEL
LIN {X 0,Y 347.814,Z 86.641,A -85,B 0,C 180,E1 -13839.909,E2 -13839.909} C_VEL
LIN {X 0,Y 347.867,Z 86.628,A -85,B 0,C 180,E1 -13842.359,E2 -13842.359} C_VEL
LIN {X 0,Y 347.898,Z 86.647,A -85,B 0,C 180,E1 -13845.97,E2 -13845.97} C_VEL
LIN {X 0,Y 347.929,Z 86.618,A -85,B 0,C 180,E1 -13849.525,E2 -13849.525} C_VEL
LIN {X 0,Y 348.075,Z 86.606,A -85,B 0,C 180,E1 -13851.874,E2 -13851.874} C_VEL
LIN {X 0,Y 348.071,Z 86.627,A -85,B 0,C 180,E1 -13854.205,E2 -13854.205} C_VEL
LIN {X 0,Y 348.206,Z 86.599,A -85,B 0,C 180,E1 -13857.686,E2 -13857.686} C_VEL
LIN {X 0,Y 348.325,Z 86.564,A -85,B 0,C 180,E1 -13859.999,E2 -13859.999} C_VEL
LIN {X 0,Y 348.206,Z 86.598,A -85,B 0,C 180,E1 -13862.313,E2 -13862.313} C_VEL
LIN {X 0,Y 348.106,Z 86.617,A -85,B 0,C 180,E1 -13866.957,E2 -13866.957} C_VEL
LIN {X 0,Y 347.968,Z 86.612,A -85,B 0,C 180,E1 -13869.298,E2 -13869.298} C_VEL
LIN {X 0,Y 347.893,Z 86.643,A -85,B 0,C 180,E1 -13872.839,E2 -13872.839} C_VEL
LIN {X 0,Y 347.838,Z 86.65,A -85,B 0,C 180,E1 -13876.431,E2 -13876.431} C_VEL
LIN {X 0,Y 347.849,Z 86.628,A -85,B 0,C 180,E1 -13878.86,E2 -13878.86} C_VEL
LIN {X 0,Y 347.774,Z 86.662,A -85,B 0,C 180,E1 -13882.579,E2 -13882.579} C_VEL
LIN {X 0,Y 347.81,Z 86.653,A -85,B 0,C 180,E1 -13885.108,E2 -13885.108} C_VEL
LIN {X 0,Y 347.806,Z 86.64,A -85,B 0,C 180,E1 -13887.693,E2 -13887.693} C_VEL
LIN {X 0,Y 347.747,Z 86.666,A -85,B 0,C 180,E1 -13890.347,E2 -13890.347} C_VEL
LIN {X 0,Y 347.745,Z 86.652,A -85,B 0,C 180,E1 -13894.043,E2 -13894.043} C_VEL
LIN {X 0,Y 347.76,Z 86.667,A -85,B 0,C 180,E1 -13897.32,E2 -13897.32} C_VEL
LIN {X 0,Y 347.752,Z 86.655,A -85,B 0,C 180,E1 -13900.293,E2 -13900.293} C_VEL
LIN {X 0,Y 347.726,Z 86.67,A -85,B 0,C 180,E1 -13903.407,E2 -13903.407} C_VEL
LIN {X 0,Y 347.721,Z 86.636,A -85,B 0,C 180,E1 -13906.686,E2 -13906.686} C_VEL
LIN {X 0,Y 347.744,Z 86.653,A -85,B 0,C 180,E1 -13910.173,E2 -13910.173} C_VEL
LIN {X 0,Y 347.759,Z 86.665,A -85,B 0,C 180,E1 -13912.679,E2 -13912.679} C_VEL
LIN {X 0,Y 347.744,Z 86.641,A -85,B 0,C 180,E1 -13915.956,E2 -13915.956} C_VEL
LIN {X 0,Y 347.745,Z 86.655,A -85,B 0,C 180,E1 -13919.652,E2 -13919.652} C_VEL
LIN {X 0,Y 347.827,Z 86.661,A -85,B 0,C 180,E1 -13923.608,E2 -13923.608} C_VEL
LIN {X 0,Y 347.785,Z 86.666,A -85,B 0,C 180,E1 -13926.162,E2 -13926.162} C_VEL
LIN {X 0,Y 347.822,Z 86.782,A -85,B 0,C 180,E1 -13929.138,E2 -13929.138} C_VEL
LIN {X 0,Y 348.019,Z 87.795,A -85,B 0,C 180,E1 -13929.459,E2 -13929.459} C_VEL
LIN {X 0,Y 349.598,Z 90.589,A -85,B 0,C 180,E1 -13929.907,E2 -13929.907} C_VEL
LIN {X 0,Y 351.805,Z 92.411,A -85,B 0,C 180,E1 -13930.407,E2 -13930.407} C_VEL
LIN {X 0,Y 353.933,Z 95.736,A -85,B 0,C 180,E1 -13930.994,E2 -13930.994} C_VEL
LIN {X 0,Y 356.535,Z 98.13,A -85,B 0,C 180,E1 -13931.644,E2 -13931.644} C_VEL
LIN {X 0,Y 359.05,Z 101.5,A -85,B 0,C 180,E1 -13932.356,E2 -13932.356} C_VEL
LIN {X 0,Y 361.876,Z 104.042,A -85,B 0,C 180,E1 -13933.127,E2 -13933.127} C_VEL
LIN {X 0,Y 364.51,Z 107.262,A -85,B 0,C 180,E1 -13933.938,E2 -13933.938} C_VEL
LIN {X 0,Y 368.034,Z 110.225,A -85,B 0,C 180,E1 -13935.004,E2 -13935.004} C_VEL
LIN {X 0,Y 371.142,Z 113.814,A -85,B 0,C 180,E1 -13936.082,E2 -13936.082} C_VEL
LIN {X 0,Y 374.487,Z 116.436,A -85,B 0,C 180,E1 -13937.295,E2 -13937.295} C_VEL
LIN {X 0,Y 377.299,Z 119.677,A -85,B 0,C 180,E1 -13938.459,E2 -13938.459} C_VEL
LIN {X 0,Y 380.198,Z 121.941,A -85,B 0,C 180,E1 -13939.73,E2 -13939.73} C_VEL
LIN {X 0,Y 382.426,Z 123.251,A -85,B 0,C 180,E1 -13940.794,E2 -13940.794} C_VEL
LIN {X 0,Y 385.153,Z 126.558,A -85,B 0,C 180,E1 -13942.452,E2 -13942.452} C_VEL
LIN {X 0,Y 387.586,Z 128.484,A -85,B 0,C 180,E1 -13944.253,E2 -13944.253} C_VEL
LIN {X 0,Y 389.26,Z 129.373,A -85,B 0,C 180,E1 -13945.859,E2 -13945.859} C_VEL
LIN {X 0,Y 390.396,Z 129.749,A -85,B 0,C 180,E1 -13947.439,E2 -13947.439} C_VEL
LIN {X 0,Y 390.991,Z 130.212,A -85,B 0,C 180,E1 -13948.97,E2 -13948.97} C_VEL
LIN {X 0,Y 391.134,Z 130.115,A -85,B 0,C 180,E1 -13950,E2 -13950} C_VEL
LIN {X 0,Y 390.861,Z 130.064,A -85,B 0,C 180,E1 -13951.546,E2 -13951.546} C_VEL
LIN {X 0,Y 390.115,Z 129.609,A -85,B 0,C 180,E1 -13953.098,E2 -13953.098} C_VEL
LIN {X 0,Y 388.503,Z 129.026,A -85,B 0,C 180,E1 -13954.929,E2 -13954.929} C_VEL
LIN {X 0,Y 386.383,Z 127.647,A -85,B 0,C 180,E1 -13956.668,E2 -13956.668} C_VEL
LIN {X 0,Y 384.174,Z 125.559,A -85,B 0,C 180,E1 -13958.143,E2 -13958.143} C_VEL
LIN {X 0,Y 382.054,Z 122.873,A -85,B 0,C 180,E1 -13959.396,E2 -13959.396} C_VEL
LIN {X 0,Y 378.834,Z 120.984,A -85,B 0,C 180,E1 -13960.894,E2 -13960.894} C_VEL
LIN {X 0,Y 375.551,Z 117.777,A -85,B 0,C 180,E1 -13962.291,E2 -13962.291} C_VEL
LIN {X 0,Y 373.856,Z 115.855,A -85,B 0,C 180,E1 -13962.942,E2 -13962.942} C_VEL
LIN {X 0,Y 370.642,Z 113.344,A -85,B 0,C 180,E1 -13964.084,E2 -13964.084} C_VEL
LIN {X 0,Y 367.17,Z 109.331,A -85,B 0,C 180,E1 -13965.274,E2 -13965.274} C_VEL
LIN {X 0,Y 363.526,Z 106.217,A -85,B 0,C 180,E1 -13966.371,E2 -13966.371} C_VEL
LIN {X 0,Y 360.956,Z 103.095,A -85,B 0,C 180,E1 -13967.125,E2 -13967.125} C_VEL
LIN {X 0,Y 358.146,Z 100.482,A -85,B 0,C 180,E1 -13967.904,E2 -13967.904} C_VEL
LIN {X 0,Y 356.109,Z 97.569,A -85,B 0,C 180,E1 -13968.466,E2 -13968.466} C_VEL
LIN {X 0,Y 353.298,Z 94.961,A -85,B 0,C 180,E1 -13969.174,E2 -13969.174} C_VEL
LIN {X 0,Y 351.282,Z 91.914,A -85,B 0,C 180,E1 -13969.718,E2 -13969.718} C_VEL
LIN {X 0,Y 349.024,Z 89.879,A -85,B 0,C 180,E1 -13970.231,E2 -13970.231} C_VEL
LIN {X 0,Y 347.918,Z 87.335,A -85,B 0,C 180,E1 -13970.624,E2 -13970.624} C_VEL
LIN {X 0,Y 347.812,Z 86.699,A -85,B 0,C 180,E1 -13971.018,E2 -13971.018} C_VEL
LIN {X 0,Y 347.809,Z 86.662,A -85,B 0,C 180,E1 -13975.109,E2 -13975.109} C_VEL
LIN {X 0,Y 347.804,Z 86.657,A -85,B 0,C 180,E1 -13977.694,E2 -13977.694} C_VEL
LIN {X 0,Y 347.746,Z 86.655,A -85,B 0,C 180,E1 -13980.348,E2 -13980.348} C_VEL
LIN {X 0,Y 347.744,Z 86.639,A -85,B 0,C 180,E1 -13984.044,E2 -13984.044} C_VEL
LIN {X 0,Y 347.759,Z 86.665,A -85,B 0,C 180,E1 -13987.321,E2 -13987.321} C_VEL
LIN {X 0,Y 347.728,Z 86.646,A -85,B 0,C 180,E1 -13990.297,E2 -13990.297} C_VEL
LIN {X 0,Y 347.719,Z 86.638,A -85,B 0,C 180,E1 -13993.409,E2 -13993.409} C_VEL
LIN {X 0,Y 347.729,Z 86.669,A -85,B 0,C 180,E1 -13996.685,E2 -13996.685} C_VEL
LIN {X 0,Y 347.755,Z 86.659,A -85,B 0,C 180,E1 -14000.171,E2 -14000.171} C_VEL
LIN {X 0,Y 347.768,Z 86.659,A -85,B 0,C 180,E1 -14003.935,E2 -14003.935} C_VEL
LIN {X 0,Y 347.73,Z 86.66,A -85,B 0,C 180,E1 -14006.928,E2 -14006.928} C_VEL
LIN {X 0,Y 347.739,Z 86.666,A -85,B 0,C 180,E1 -14009.545,E2 -14009.545} C_VEL
LIN {X 0,Y 347.126,Z 86.745,A -85,B 0,C 180,E1 -14010.512,E2 -14010.512} C_VEL
LIN {X 0,Y 344.308,Z 87.089,A -85,B 0,C 180,E1 -14012.088,E2 -14012.088} C_VEL
LIN {X 0,Y 341.889,Z 87.383,A -85,B 0,C 180,E1 -14013.363,E2 -14013.363} C_VEL
LIN {X 0,Y 340.845,Z 87.515,A -85,B 0,C 180,E1 -14014.349,E2 -14014.349} C_VEL
LIN {X 0,Y 340.759,Z 87.528,A -85,B 0,C 180,E1 -14014.683,E2 -14014.683} C_VEL
LIN {X 0,Y 340.739,Z 87.539,A -85,B 0,C 180,E1 -14018.207,E2 -14018.207} C_VEL
LIN {X 0,Y 340.856,Z 87.503,A -85,B 0,C 180,E1 -14021.985,E2 -14021.985} C_VEL
LIN {X 0,Y 340.868,Z 87.523,A -85,B 0,C 180,E1 -14025.706,E2 -14025.706} C_VEL
LIN {X 0,Y 340.873,Z 87.498,A -85,B 0,C 180,E1 -14029.307,E2 -14029.307} C_VEL
LIN {X 0,Y 341.075,Z 87.493,A -85,B 0,C 180,E1 -14032.899,E2 -14032.899} C_VEL
LIN {X 0,Y 341.167,Z 87.475,A -85,B 0,C 180,E1 -14037.639,E2 -14037.639} C_VEL
LIN {X 0,Y 341.275,Z 87.442,A -85,B 0,C 180,E1 -14040.001,E2 -14040.001} C_VEL
LIN {X 0,Y 341.168,Z 87.476,A -85,B 0,C 180,E1 -14042.362,E2 -14042.362} C_VEL
LIN {X 0,Y 341.078,Z 87.492,A -85,B 0,C 180,E1 -14047.102,E2 -14047.102} C_VEL
LIN {X 0,Y 340.871,Z 87.498,A -85,B 0,C 180,E1 -14050.694,E2 -14050.694} C_VEL
LIN {X 0,Y 340.864,Z 87.522,A -85,B 0,C 180,E1 -14054.325,E2 -14054.325} C_VEL
LIN {X 0,Y 340.838,Z 87.498,A -85,B 0,C 180,E1 -14058.467,E2 -14058.467} C_VEL
LIN {X 0,Y 340.755,Z 87.536,A -85,B 0,C 180,E1 -14061.857,E2 -14061.857} C_VEL
LIN {X 0,Y 340.773,Z 87.52,A -85,B 0,C 180,E1 -14065.665,E2 -14065.665} C_VEL
LIN {X 0,Y 340.729,Z 87.528,A -85,B 0,C 180,E1 -14068.321,E2 -14068.321} C_VEL
LIN {X 0,Y 340.699,Z 87.548,A -85,B 0,C 180,E1 -14071.045,E2 -14071.045} C_VEL
LIN {X 0,Y 340.719,Z 87.531,A -85,B 0,C 180,E1 -14075.279,E2 -14075.279} C_VEL
LIN {X 0,Y 340.711,Z 87.544,A -85,B 0,C 180,E1 -14078.387,E2 -14078.387} C_VEL
LIN {X 0,Y 340.7,Z 87.544,A -85,B 0,C 180,E1 -14082.046,E2 -14082.046} C_VEL
LIN {X 0,Y 340.654,Z 87.55,A -85,B 0,C 180,E1 -14086.227,E2 -14086.227} C_VEL
LIN {X 0,Y 340.689,Z 87.521,A -85,B 0,C 180,E1 -14089.754,E2 -14089.754} C_VEL
LIN {X 0,Y 340.709,Z 87.541,A -85,B 0,C 180,E1 -14093.259,E2 -14093.259} C_VEL
LIN {X 0,Y 340.734,Z 87.547,A -85,B 0,C 180,E1 -14097.219,E2 -14097.219} C_VEL
LIN {X 0,Y 342.014,Z 93.828,A -85,B 0,C 180,E1 -14099.662,E2 -14099.662} C_VEL
LIN {X 0,Y 343.693,Z 102.522,A -85,B 0,C 180,E1 -14102.607,E2 -14102.607} C_VEL
LIN {X 0,Y 343.991,Z 106.698,A -85,B 0,C 180,E1 -14104.022,E2 -14104.022} C_VEL
LIN {X 0,Y 343.04,Z 114.205,A -85,B 0,C 180,E1 -14106.407,E2 -14106.407} C_VEL
LIN {X 0,Y 343.473,Z 116.686,A -85,B 0,C 180,E1 -14106.571,E2 -14106.571} C_VEL
LIN {X 0,Y 348.209,Z 139.808,A -85,B 0,C 180,E1 -14107.412,E2 -14107.412} C_VEL
LIN {X 0,Y 350.17,Z 151.369,A -85,B 0,C 180,E1 -14107.795,E2 -14107.795} C_VEL
LIN {X 0,Y 349.036,Z 219.126,A -85,B 0,C 180,E1 -14109.214,E2 -14109.214} C_VEL
LIN {X 0,Y 348.511,Z 229.869,A -85,B 0,C 180,E1 -14109.567,E2 -14109.567} C_VEL
LIN {X 0,Y 347.865,Z 238.969,A -85,B 0,C 180,E1 -14109.99,E2 -14109.99} C_VEL
LIN {X 0,Y 347.089,Z 248.323,A -85,B 0,C 180,E1 -14110.559,E2 -14110.559} C_VEL
LIN {X 0,Y 346.14,Z 258.463,A -85,B 0,C 180,E1 -14111.35,E2 -14111.35} C_VEL
LIN {X 0,Y 345.121,Z 267.458,A -85,B 0,C 180,E1 -14112.214,E2 -14112.214} C_VEL
LIN {X 0,Y 344.064,Z 276.184,A -85,B 0,C 180,E1 -14113.23,E2 -14113.23} C_VEL
LIN {X 0,Y 343.103,Z 283.943,A -85,B 0,C 180,E1 -14114.31,E2 -14114.31} C_VEL
LIN {X 0,Y 342.319,Z 290.8,A -85,B 0,C 180,E1 -14115.434,E2 -14115.434} C_VEL
LIN {X 0,Y 341.585,Z 297.003,A -85,B 0,C 180,E1 -14116.617,E2 -14116.617} C_VEL
LIN {X 0,Y 340.7,Z 303.538,A -85,B 0,C 180,E1 -14118.096,E2 -14118.096} C_VEL
LIN {X 0,Y 340.219,Z 308.041,A -85,B 0,C 180,E1 -14119.286,E2 -14119.286} C_VEL
LIN {X 0,Y 339.652,Z 313.534,A -85,B 0,C 180,E1 -14121.072,E2 -14121.072} C_VEL
LIN {X 0,Y 339.275,Z 317.859,A -85,B 0,C 180,E1 -14122.86,E2 -14122.86} C_VEL
LIN {X 0,Y 339.134,Z 320.323,A -85,B 0,C 180,E1 -14124.116,E2 -14124.116} C_VEL
LIN {X 0,Y 339.066,Z 323.415,A -85,B 0,C 180,E1 -14126.435,E2 -14126.435} C_VEL
LIN {X 0,Y 338.998,Z 324.472,A -85,B 0,C 180,E1 -14127.624,E2 -14127.624} C_VEL
LIN {X 0,Y 339.007,Z 325.061,A -85,B 0,C 180,E1 -14128.812,E2 -14128.812} C_VEL
LIN {X 0,Y 339.068,Z 325.217,A -85,B 0,C 180,E1 -14130,E2 -14130} C_VEL
LIN {X 0,Y 339.007,Z 325.061,A -85,B 0,C 180,E1 -14131.188,E2 -14131.188} C_VEL
LIN {X 0,Y 338.998,Z 324.472,A -85,B 0,C 180,E1 -14132.376,E2 -14132.376} C_VEL
LIN {X 0,Y 339.062,Z 322.026,A -85,B 0,C 180,E1 -14134.756,E2 -14134.756} C_VEL
LIN {X 0,Y 339.178,Z 319.075,A -85,B 0,C 180,E1 -14136.544,E2 -14136.544} C_VEL
LIN {X 0,Y 339.511,Z 315.088,A -85,B 0,C 180,E1 -14138.332,E2 -14138.332} C_VEL
LIN {X 0,Y 339.983,Z 309.957,A -85,B 0,C 180,E1 -14140.12,E2 -14140.12} C_VEL
LIN {X 0,Y 340.54,Z 304.693,A -85,B 0,C 180,E1 -14141.608,E2 -14141.608} C_VEL
LIN {X 0,Y 341.399,Z 298.379,A -85,B 0,C 180,E1 -14143.088,E2 -14143.088} C_VEL
LIN {X 0,Y 342.124,Z 292.427,A -85,B 0,C 180,E1 -14144.271,E2 -14144.271} C_VEL
LIN {X 0,Y 343.168,Z 284.454,A -85,B 0,C 180,E1 -14145.607,E2 -14145.607} C_VEL
LIN {X 0,Y 344.237,Z 275.051,A -85,B 0,C 180,E1 -14146.914,E2 -14146.914} C_VEL
LIN {X 0,Y 345.454,Z 264.755,A -85,B 0,C 180,E1 -14148.074,E2 -14148.074} C_VEL
LIN {X 0,Y 346.738,Z 252.351,A -85,B 0,C 180,E1 -14149.154,E2 -14149.154} C_VEL
LIN {X 0,Y 347.693,Z 241.544,A -85,B 0,C 180,E1 -14149.867,E2 -14149.867} C_VEL
LIN {X 0,Y 348.41,Z 231.617,A -85,B 0,C 180,E1 -14150.363,E2 -14150.363} C_VEL
LIN {X 0,Y 348.899,Z 221.762,A -85,B 0,C 180,E1 -14150.718,E2 -14150.718} C_VEL
LIN {X 0,Y 349.484,Z 197.95,A -85,B 0,C 180,E1 -14151.243,E2 -14151.243} C_VEL
LIN {X 0,Y 350.236,Z 151.836,A -85,B 0,C 180,E1 -14152.191,E2 -14152.191} C_VEL
LIN {X 0,Y 345.802,Z 127.244,A -85,B 0,C 180,E1 -14153.03,E2 -14153.03} C_VEL
LIN {X 0,Y 343.052,Z 114.484,A -85,B 0,C 180,E1 -14153.547,E2 -14153.547} C_VEL
LIN {X 0,Y 343.258,Z 112.263,A -85,B 0,C 180,E1 -14154.173,E2 -14154.173} C_VEL
LIN {X 0,Y 344.061,Z 105.85,A -85,B 0,C 180,E1 -14156.255,E2 -14156.255} C_VEL
LIN {X 0,Y 343.244,Z 99.872,A -85,B 0,C 180,E1 -14158.304,E2 -14158.304} C_VEL
LIN {X 0,Y 341.379,Z 90.509,A -85,B 0,C 180,E1 -14161.618,E2 -14161.618} C_VEL
LIN {X 0,Y 340.734,Z 87.551,A -85,B 0,C 180,E1 -14162.781,E2 -14162.781} C_VEL
LIN {X 0,Y 340.709,Z 87.541,A -85,B 0,C 180,E1 -14166.741,E2 -14166.741} C_VEL
LIN {X 0,Y 340.689,Z 87.521,A -85,B 0,C 180,E1 -14170.246,E2 -14170.246} C_VEL
LIN {X 0,Y 340.654,Z 87.551,A -85,B 0,C 180,E1 -14173.773,E2 -14173.773} C_VEL
LIN {X 0,Y 340.7,Z 87.545,A -85,B 0,C 180,E1 -14177.954,E2 -14177.954} C_VEL
LIN {X 0,Y 340.734,Z 87.541,A -85,B 0,C 180,E1 -14181.772,E2 -14181.772} C_VEL
LIN {X 0,Y 340.724,Z 87.523,A -85,B 0,C 180,E1 -14185.595,E2 -14185.595} C_VEL
LIN {X 0,Y 340.699,Z 87.548,A -85,B 0,C 180,E1 -14188.955,E2 -14188.955} C_VEL
LIN {X 0,Y 340.804,Z 87.509,A -85,B 0,C 180,E1 -14193.019,E2 -14193.019} C_VEL
LIN {X 0,Y 340.731,Z 87.541,A -85,B 0,C 180,E1 -14196.927,E2 -14196.927} C_VEL
LIN {X 0,Y 340.792,Z 87.505,A -85,B 0,C 180,E1 -14200.733,E2 -14200.733} C_VEL
LIN {X 0,Y 340.788,Z 87.523,A -85,B 0,C 180,E1 -14203.218,E2 -14203.218} C_VEL
LIN {X 0,Y 340.845,Z 87.521,A -85,B 0,C 180,E1 -14206.89,E2 -14206.89} C_VEL
LIN {X 0,Y 340.929,Z 87.485,A -85,B 0,C 180,E1 -14210.507,E2 -14210.507} C_VEL
LIN {X 0,Y 341.078,Z 87.492,A -85,B 0,C 180,E1 -14212.898,E2 -14212.898} C_VEL
LIN {X 0,Y 341.168,Z 87.476,A -85,B 0,C 180,E1 -14217.638,E2 -14217.638} C_VEL
LIN {X 0,Y 341.275,Z 87.442,A -85,B 0,C 180,E1 -14219.999,E2 -14219.999} C_VEL
LIN {X 0,Y 341.167,Z 87.475,A -85,B 0,C 180,E1 -14222.361,E2 -14222.361} C_VEL
LIN {X 0,Y 341.075,Z 87.493,A -85,B 0,C 180,E1 -14227.101,E2 -14227.101} C_VEL
LIN {X 0,Y 340.873,Z 87.498,A -85,B 0,C 180,E1 -14230.693,E2 -14230.693} C_VEL
LIN {X 0,Y 340.862,Z 87.524,A -85,B 0,C 180,E1 -14234.324,E2 -14234.324} C_VEL
LIN {X 0,Y 340.835,Z 87.503,A -85,B 0,C 180,E1 -14238.466,E2 -14238.466} C_VEL
LIN {X 0,Y 340.752,Z 87.537,A -85,B 0,C 180,E1 -14241.856,E2 -14241.856} C_VEL
LIN {X 0,Y 340.77,Z 87.524,A -85,B 0,C 180,E1 -14245.664,E2 -14245.664} C_VEL
LIN {X 0,Y 340.726,Z 87.526,A -85,B 0,C 180,E1 -14248.32,E2 -14248.32} C_VEL
LIN {X 0,Y 340.695,Z 87.549,A -85,B 0,C 180,E1 -14251.044,E2 -14251.044} C_VEL
LIN {X 0,Y 340.716,Z 87.531,A -85,B 0,C 180,E1 -14255.278,E2 -14255.278} C_VEL
LIN {X 0,Y 340.715,Z 87.547,A -85,B 0,C 180,E1 -14258.387,E2 -14258.387} C_VEL
LIN {X 0,Y 340.726,Z 87.536,A -85,B 0,C 180,E1 -14262.051,E2 -14262.051} C_VEL
LIN {X 0,Y 340.649,Z 87.522,A -85,B 0,C 180,E1 -14266.226,E2 -14266.226} C_VEL
LIN {X 0,Y 340.684,Z 87.523,A -85,B 0,C 180,E1 -14269.753,E2 -14269.753} C_VEL
LIN {X 0,Y 340.702,Z 87.54,A -85,B 0,C 180,E1 -14273.258,E2 -14273.258} C_VEL
LIN {X 0,Y 340.688,Z 87.521,A -85,B 0,C 180,E1 -14276.153,E2 -14276.153} C_VEL
LIN {X 0,Y 340.737,Z 87.521,A -85,B 0,C 180,E1 -14280.329,E2 -14280.329} C_VEL
LIN {X 0,Y 340.8,Z 87.535,A -85,B 0,C 180,E1 -14283.02,E2 -14283.02} C_VEL
LIN {X 0,Y 340.752,Z 87.541,A -85,B 0,C 180,E1 -14285.638,E2 -14285.638} C_VEL
LIN {X 0,Y 340.749,Z 87.651,A -85,B 0,C 180,E1 -14287.813,E2 -14287.813} C_VEL
LIN {X 0,Y 340.931,Z 88.487,A -85,B 0,C 180,E1 -14288.111,E2 -14288.111} C_VEL
LIN {X 0,Y 342.359,Z 91.226,A -85,B 0,C 180,E1 -14288.51,E2 -14288.51} C_VEL
LIN {X 0,Y 344.49,Z 93.294,A -85,B 0,C 180,E1 -14288.961,E2 -14288.961} C_VEL
LIN {X 0,Y 346.725,Z 96.608,A -85,B 0,C 180,E1 -14289.518,E2 -14289.518} C_VEL
LIN {X 0,Y 348.969,Z 98.833,A -85,B 0,C 180,E1 -14290.042,E2 -14290.042} C_VEL
LIN {X 0,Y 351.593,Z 102.19,A -85,B 0,C 180,E1 -14290.687,E2 -14290.687} C_VEL
LIN {X 0,Y 353.899,Z 104.487,A -85,B 0,C 180,E1 -14291.28,E2 -14291.28} C_VEL
LIN {X 0,Y 357.171,Z 108.316,A -85,B 0,C 180,E1 -14292.137,E2 -14292.137} C_VEL
LIN {X 0,Y 359.47,Z 110.421,A -85,B 0,C 180,E1 -14292.775,E2 -14292.775} C_VEL
LIN {X 0,Y 362.8,Z 114.104,A -85,B 0,C 180,E1 -14293.735,E2 -14293.735} C_VEL
LIN {X 0,Y 365.929,Z 116.722,A -85,B 0,C 180,E1 -14294.673,E2 -14294.673} C_VEL
LIN {X 0,Y 369.295,Z 120.435,A -85,B 0,C 180,E1 -14295.807,E2 -14295.807} C_VEL
LIN {X 0,Y 372.825,Z 123.258,A -85,B 0,C 180,E1 -14297.045,E2 -14297.045} C_VEL
LIN {X 0,Y 376.27,Z 126.891,A -85,B 0,C 180,E1 -14298.427,E2 -14298.427} C_VEL
LIN {X 0,Y 379.583,Z 129.236,A -85,B 0,C 180,E1 -14299.877,E2 -14299.877} C_VEL
LIN {X 0,Y 381.145,Z 130.139,A -85,B 0,C 180,E1 -14300.617,E2 -14300.617} C_VEL
LIN {X 0,Y 383.823,Z 133.32,A -85,B 0,C 180,E1 -14302.189,E2 -14302.189} C_VEL
LIN {X 0,Y 386.288,Z 135.257,A -85,B 0,C 180,E1 -14303.895,E2 -14303.895} C_VEL
LIN {X 0,Y 388.386,Z 136.414,A -85,B 0,C 180,E1 -14305.849,E2 -14305.849} C_VEL
LIN {X 0,Y 389.529,Z 136.797,A -85,B 0,C 180,E1 -14307.434,E2 -14307.434} C_VEL
LIN {X 0,Y 390.126,Z 137.258,A -85,B 0,C 180,E1 -14308.968,E2 -14308.968} C_VEL
LIN {X 0,Y 390.27,Z 137.149,A -85,B 0,C 180,E1 -14310,E2 -14310} C_VEL
LIN {X 0,Y 389.992,Z 137.112,A -85,B 0,C 180,E1 -14311.549,E2 -14311.549} C_VEL
LIN {X 0,Y 389.238,Z 136.655,A -85,B 0,C 180,E1 -14313.105,E2 -14313.105} C_VEL
